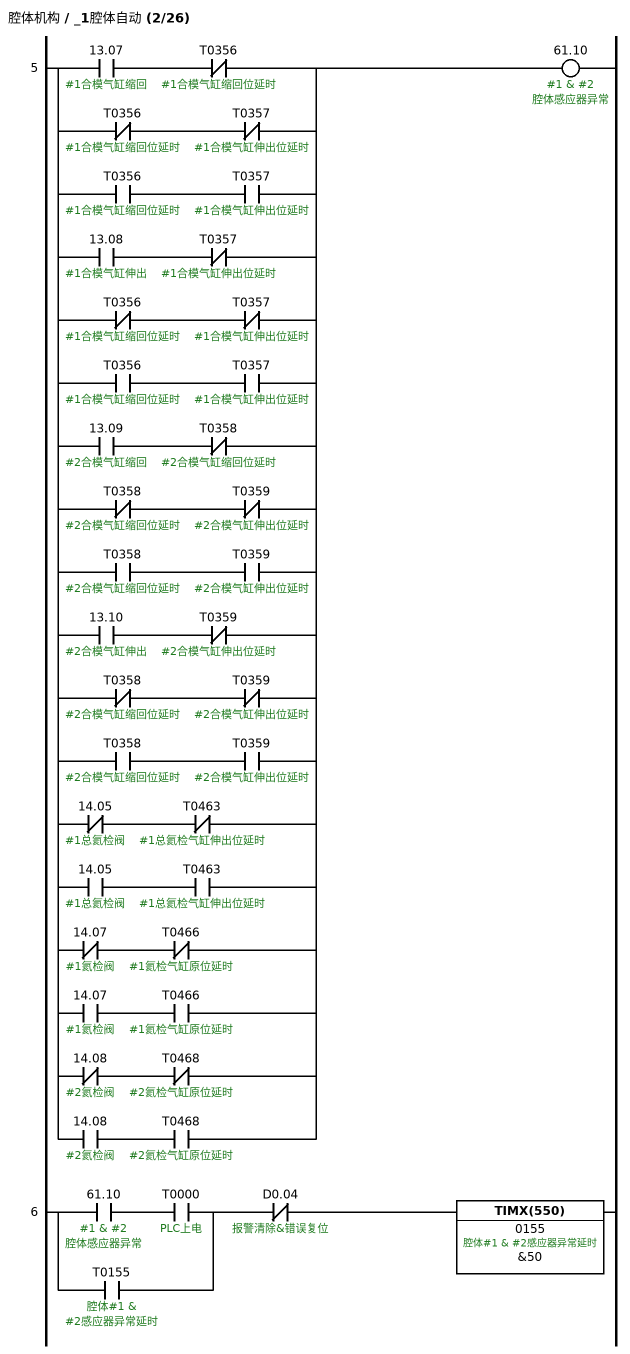
; [picture p240: 腔体机构 / _1腔体自动, rungs 5-6]
; rung 5
LD 13.07  ; #1合模气缸缩回
ANDNOT T0356  ; #1合模气缸缩回位延时
LDNOT T0356  ; #1合模气缸缩回位延时
ANDNOT T0357  ; #1合模气缸伸出位延时
ORLD
LD T0356  ; #1合模气缸缩回位延时
AND T0357  ; #1合模气缸伸出位延时
ORLD
LD 13.08  ; #1合模气缸伸出
ANDNOT T0357  ; #1合模气缸伸出位延时
ORLD
LDNOT T0356  ; #1合模气缸缩回位延时
ANDNOT T0357  ; #1合模气缸伸出位延时
ORLD
LD T0356  ; #1合模气缸缩回位延时
AND T0357  ; #1合模气缸伸出位延时
ORLD
LD 13.09  ; #2合模气缸缩回
ANDNOT T0358  ; #2合模气缸缩回位延时
ORLD
LDNOT T0358  ; #2合模气缸缩回位延时
ANDNOT T0359  ; #2合模气缸伸出位延时
ORLD
LD T0358  ; #2合模气缸缩回位延时
AND T0359  ; #2合模气缸伸出位延时
ORLD
LD 13.10  ; #2合模气缸伸出
ANDNOT T0359  ; #2合模气缸伸出位延时
ORLD
LDNOT T0358  ; #2合模气缸缩回位延时
ANDNOT T0359  ; #2合模气缸伸出位延时
ORLD
LD T0358  ; #2合模气缸缩回位延时
AND T0359  ; #2合模气缸伸出位延时
ORLD
LDNOT 14.05  ; #1总氦检阀
ANDNOT T0463  ; #1总氦检气缸伸出位延时
ORLD
LD 14.05  ; #1总氦检阀
AND T0463  ; #1总氦检气缸伸出位延时
ORLD
LDNOT 14.07  ; #1氦检阀
ANDNOT T0466  ; #1氦检气缸原位延时
ORLD
LD 14.07  ; #1氦检阀
AND T0466  ; #1氦检气缸原位延时
ORLD
LDNOT 14.08  ; #2氦检阀
ANDNOT T0468  ; #2氦检气缸原位延时
ORLD
LD 14.08  ; #2氦检阀
AND T0468  ; #2氦检气缸原位延时
ORLD
OUT 61.10  ; #1 & #2 腔体感应器异常
; rung 6
LD 61.10  ; #1 & #2 腔体感应器异常
AND T0000  ; PLC上电
OR T0155  ; 腔体#1 & #2感应器异常延时
ANDNOT D0.04  ; 报警清除&错误复位
TIMX(550) 0155 &50  ; 腔体#1 & #2感应器异常延时

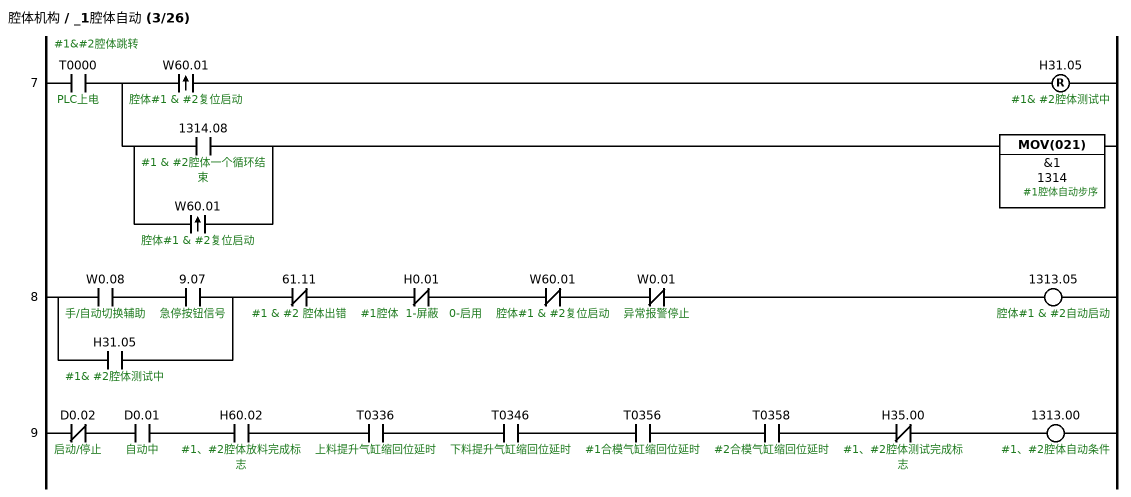
; rung 7: #1&#2腔体跳转
LD T0000  ; PLC上电
OUT TR0
@AND W60.01  ; 腔体#1 & #2复位启动
RSET H31.05  ; #1& #2腔体测试中
LD TR0
LD 1314.08  ; #1 & #2腔体一个循环结束
@OR W60.01  ; 腔体#1 & #2复位启动
ANDLD
MOV(021) &1 1314  ; #1腔体自动步序
; rung 8
LD W0.08  ; 手/自动切换辅助
AND 9.07  ; 急停按钮信号
OR H31.05  ; #1& #2腔体测试中
ANDNOT 61.11  ; #1 & #2 腔体出错
ANDNOT H0.01  ; #1腔体  1-屏蔽   0-启用
ANDNOT W60.01  ; 腔体#1 & #2复位启动
ANDNOT W0.01  ; 异常报警停止
OUT 1313.05  ; 腔体#1 & #2自动启动
; rung 9
LDNOT D0.02  ; 启动/停止
AND D0.01  ; 自动中
AND H60.02  ; #1、#2腔体放料完成标志
AND T0336  ; 上料提升气缸缩回位延时
AND T0346  ; 下料提升气缸缩回位延时
AND T0356  ; #1合模气缸缩回位延时
AND T0358  ; #2合模气缸缩回位延时
ANDNOT H35.00  ; #1、#2腔体测试完成标志
OUT 1313.00  ; #1、#2腔体自动条件

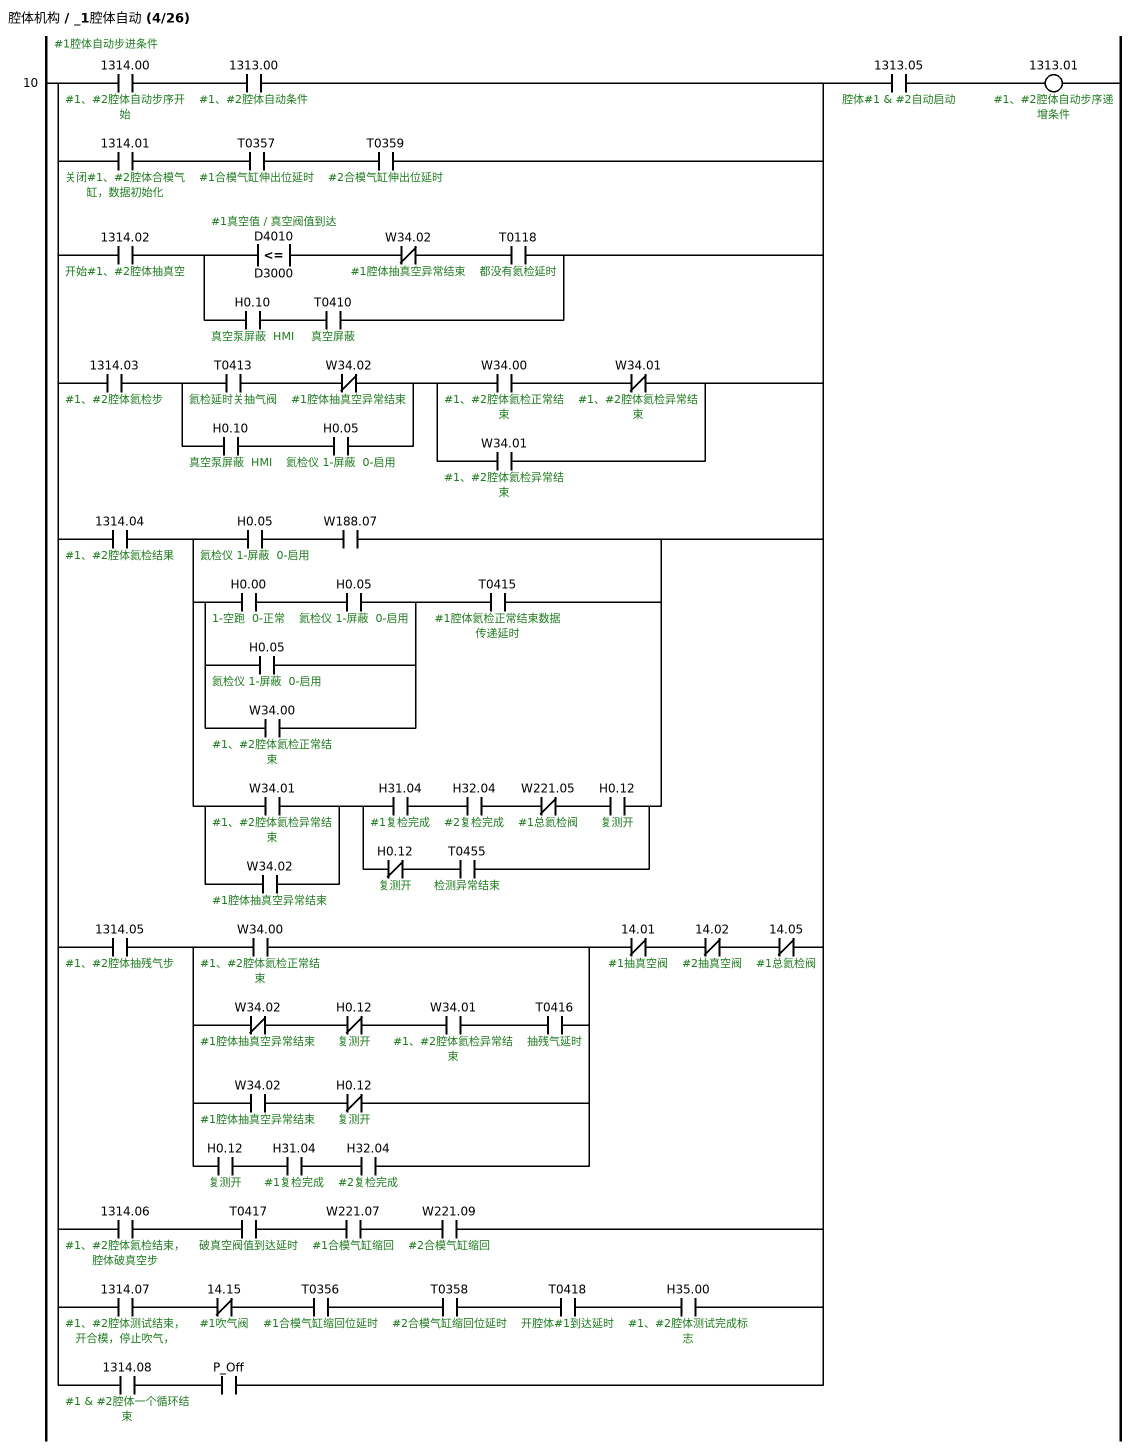
; rung 10: #1腔体自动步进条件
LD 1314.00  ; #1、#2腔体自动步序开始
AND 1313.00  ; #1、#2腔体自动条件
LD 1314.01  ; 关闭#1、#2腔体合模气缸，数据初始化
AND T0357  ; #1合模气缸伸出位延时
AND T0359  ; #2合模气缸伸出位延时
ORLD
LD 1314.02  ; 开始#1、#2腔体抽真空
LD<=F(332) D4010 D3000  ; #1真空值, 真空阀值到达
ANDNOT W34.02  ; #1腔体抽真空异常结束
AND T0118  ; 都没有氦检延时
LD H0.10  ; 真空泵屏蔽  HMI
AND T0410  ; 真空屏蔽
ORLD
ANDLD
ORLD
LD 1314.03  ; #1、#2腔体氦检步
LD T0413  ; 氦检延时关抽气阀
ANDNOT W34.02  ; #1腔体抽真空异常结束
LD H0.10  ; 真空泵屏蔽  HMI
AND H0.05  ; 氦检仪 1-屏蔽  0-启用
ORLD
ANDLD
LD W34.00  ; #1、#2腔体氦检正常结束
ANDNOT W34.01  ; #1、#2腔体氦检异常结束
OR W34.01  ; #1、#2腔体氦检异常结束
ANDLD
ORLD
LD 1314.04  ; #1、#2腔体氦检结果
LD H0.05  ; 氦检仪 1-屏蔽  0-启用
AND W188.07
LD H0.00  ; 1-空跑  0-正常
AND H0.05  ; 氦检仪 1-屏蔽  0-启用
OR H0.05  ; 氦检仪 1-屏蔽  0-启用
OR W34.00  ; #1、#2腔体氦检正常结束
AND T0415  ; #1腔体氦检正常结束数据传递延时
ORLD
LD W34.01  ; #1、#2腔体氦检异常结束
OR W34.02  ; #1腔体抽真空异常结束
LD H31.04  ; #1复检完成
AND H32.04  ; #2复检完成
ANDNOT W221.05  ; #1总氦检阀
AND H0.12  ; 复测开
LDNOT H0.12  ; 复测开
AND T0455  ; 检测异常结束
ORLD
ANDLD
ORLD
ANDLD
ORLD
LD 1314.05  ; #1、#2腔体抽残气步
LD W34.00  ; #1、#2腔体氦检正常结束
LDNOT W34.02  ; #1腔体抽真空异常结束
ANDNOT H0.12  ; 复测开
AND W34.01  ; #1、#2腔体氦检异常结束
AND T0416  ; 抽残气延时
ORLD
LD W34.02  ; #1腔体抽真空异常结束
ANDNOT H0.12  ; 复测开
ORLD
LD H0.12  ; 复测开
AND H31.04  ; #1复检完成
AND H32.04  ; #2复检完成
ORLD
ANDLD
ANDNOT 14.01  ; #1抽真空阀
ANDNOT 14.02  ; #2抽真空阀
ANDNOT 14.05  ; #1总氦检阀
ORLD
LD 1314.06  ; #1、#2腔体氦检结束，腔体破真空步
AND T0417  ; 破真空阀值到达延时
AND W221.07  ; #1合模气缸缩回
AND W221.09  ; #2合模气缸缩回
ORLD
LD 1314.07  ; #1、#2腔体测试结束，开合模，停止吹气，
ANDNOT 14.15  ; #1吹气阀
AND T0356  ; #1合模气缸缩回位延时
AND T0358  ; #2合模气缸缩回位延时
AND T0418  ; 开腔体#1到达延时
AND H35.00  ; #1、#2腔体测试完成标志
ORLD
LD 1314.08  ; #1 & #2腔体一个循环结束
AND P_Off
ORLD
AND 1313.05  ; 腔体#1 & #2自动启动
OUT 1313.01  ; #1、#2腔体自动步序递增条件

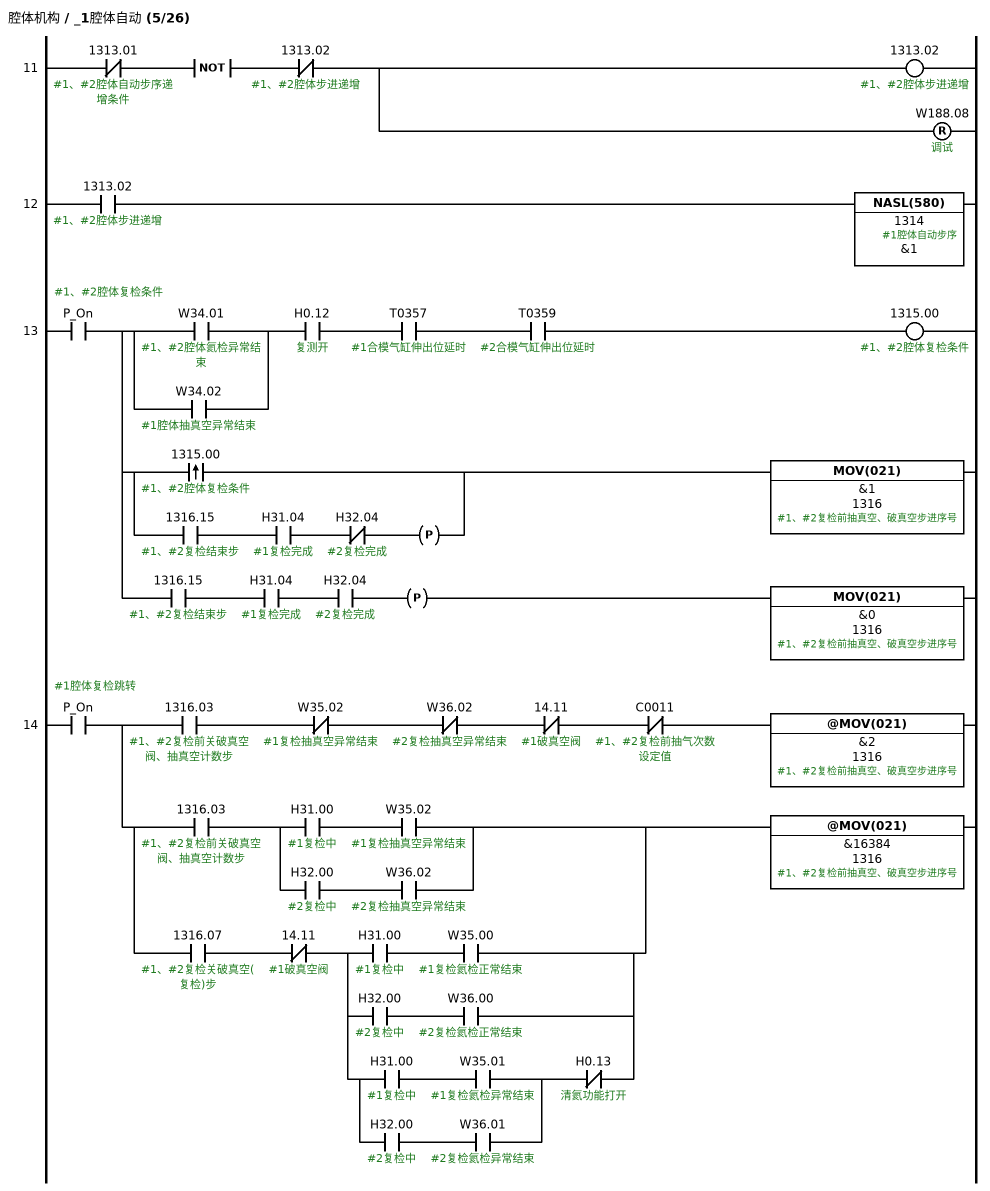
; rung 11
LDNOT 1313.01  ; #1、#2腔体自动步序递增条件
NOT(520)
ANDNOT 1313.02  ; #1、#2腔体步进递增
OUT 1313.02  ; #1、#2腔体步进递增
RSET W188.08  ; 调试
; rung 12
LD 1313.02  ; #1、#2腔体步进递增
NASL(580) 1314 &1  ; #1腔体自动步序
; rung 13: #1、#2腔体复检条件
LD P_On
OUT TR0
LD W34.01  ; #1、#2腔体氦检异常结束
OR W34.02  ; #1腔体抽真空异常结束
ANDLD
AND H0.12  ; 复测开
AND T0357  ; #1合模气缸伸出位延时
AND T0359  ; #2合模气缸伸出位延时
OUT 1315.00  ; #1、#2腔体复检条件
LD TR0
@LD 1315.00  ; #1、#2腔体复检条件
LD 1316.15  ; #1、#2复检结束步
AND H31.04  ; #1复检完成
ANDNOT H32.04  ; #2复检完成
UP(521)
ORLD
ANDLD
MOV(021) &1 1316  ; #1、#2复检前抽真空、破真空步进序号
LD TR0
AND 1316.15  ; #1、#2复检结束步
AND H31.04  ; #1复检完成
AND H32.04  ; #2复检完成
UP(521)
MOV(021) &0 1316  ; #1、#2复检前抽真空、破真空步进序号
; rung 14: #1腔体复检跳转
LD P_On
OUT TR0
AND 1316.03  ; #1、#2复检前关破真空阀、抽真空计数步
ANDNOT W35.02  ; #1复检抽真空异常结束
ANDNOT W36.02  ; #2复检抽真空异常结束
ANDNOT 14.11  ; #1破真空阀
ANDNOT C0011  ; #1、#2复检前抽气次数设定值
@MOV(021) &2 1316  ; #1、#2复检前抽真空、破真空步进序号
LD TR0
LD 1316.03  ; #1、#2复检前关破真空阀、抽真空计数步
LD H31.00  ; #1复检中
AND W35.02  ; #1复检抽真空异常结束
LD H32.00  ; #2复检中
AND W36.02  ; #2复检抽真空异常结束
ORLD
ANDLD
LD 1316.07  ; #1、#2复检关破真空(复检)步
ANDNOT 14.11  ; #1破真空阀
LD H31.00  ; #1复检中
AND W35.00  ; #1复检氦检正常结束
LD H32.00  ; #2复检中
AND W36.00  ; #2复检氦检正常结束
ORLD
LD H31.00  ; #1复检中
AND W35.01  ; #1复检氦检异常结束
LD H32.00  ; #2复检中
AND W36.01  ; #2复检氦检异常结束
ORLD
ANDNOT H0.13  ; 清氦功能打开
ORLD
ANDLD
ORLD
ANDLD
@MOV(021) &16384 1316  ; #1、#2复检前抽真空、破真空步进序号

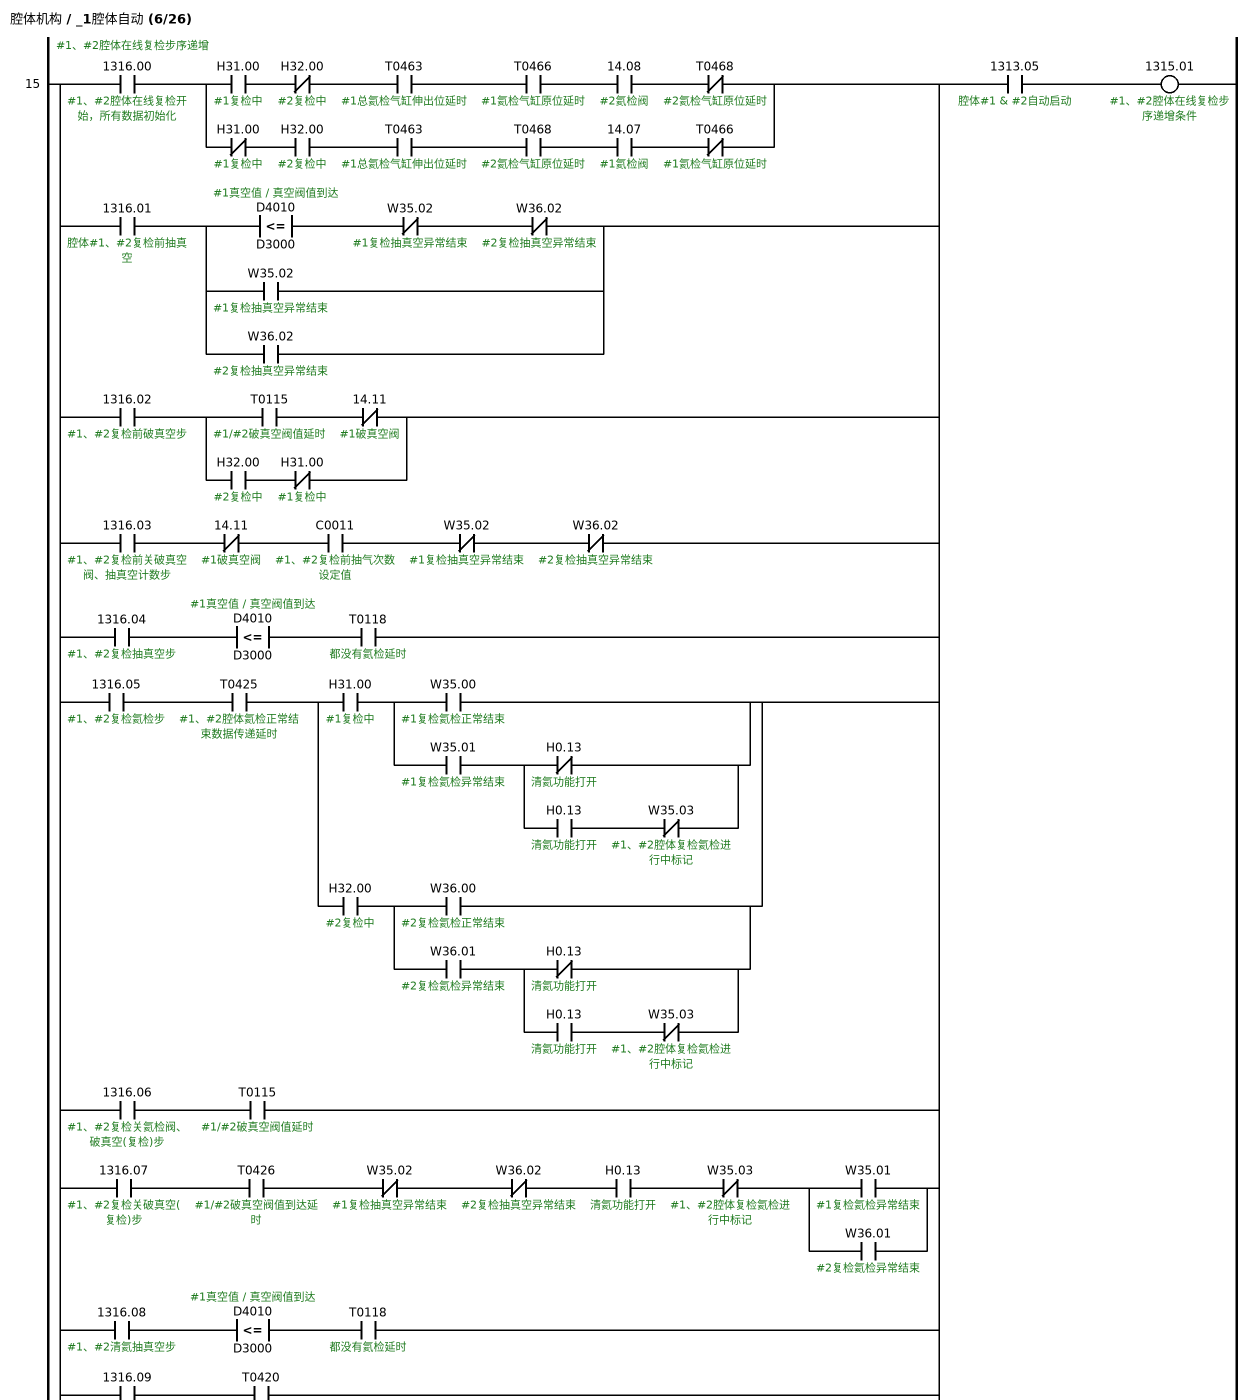

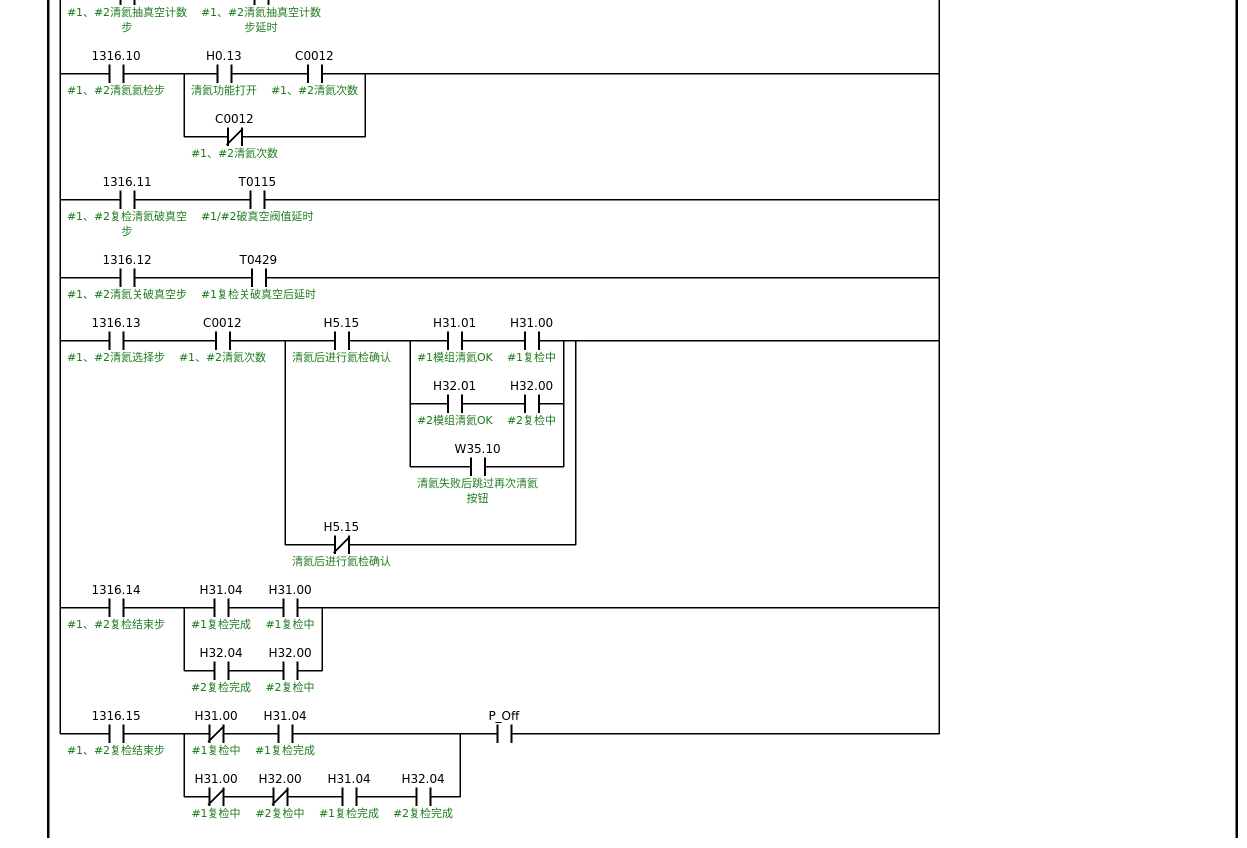
; rung 15: #1、#2腔体在线复检步序递增
LD 1316.00  ; #1、#2腔体在线复检开始，所有数据初始化
LD H31.00  ; #1复检中
ANDNOT H32.00  ; #2复检中
AND T0463  ; #1总氦检气缸伸出位延时
AND T0466  ; #1氦检气缸原位延时
AND 14.08  ; #2氦检阀
ANDNOT T0468  ; #2氦检气缸原位延时
LDNOT H31.00  ; #1复检中
AND H32.00  ; #2复检中
AND T0463  ; #1总氦检气缸伸出位延时
AND T0468  ; #2氦检气缸原位延时
AND 14.07  ; #1氦检阀
ANDNOT T0466  ; #1氦检气缸原位延时
ORLD
ANDLD
LD 1316.01  ; 腔体#1、#2复检前抽真空
LD<=F(332) D4010 D3000  ; #1真空值, 真空阀值到达
ANDNOT W35.02  ; #1复检抽真空异常结束
ANDNOT W36.02  ; #2复检抽真空异常结束
OR W35.02  ; #1复检抽真空异常结束
OR W36.02  ; #2复检抽真空异常结束
ANDLD
ORLD
LD 1316.02  ; #1、#2复检前破真空步
LD T0115  ; #1/#2破真空阀值延时
ANDNOT 14.11  ; #1破真空阀
LD H32.00  ; #2复检中
ANDNOT H31.00  ; #1复检中
ORLD
ANDLD
ORLD
LD 1316.03  ; #1、#2复检前关破真空阀、抽真空计数步
ANDNOT 14.11  ; #1破真空阀
AND C0011  ; #1、#2复检前抽气次数设定值
ANDNOT W35.02  ; #1复检抽真空异常结束
ANDNOT W36.02  ; #2复检抽真空异常结束
ORLD
LD 1316.04  ; #1、#2复检抽真空步
AND<=F(332) D4010 D3000  ; #1真空值, 真空阀值到达
AND T0118  ; 都没有氦检延时
ORLD
LD 1316.05  ; #1、#2复检氦检步
AND T0425  ; #1、#2腔体氦检正常结束数据传递延时
LD H31.00  ; #1复检中
LD W35.00  ; #1复检氦检正常结束
LD W35.01  ; #1复检氦检异常结束
LDNOT H0.13  ; 清氦功能打开
LD H0.13  ; 清氦功能打开
ANDNOT W35.03  ; #1、#2腔体复检氦检进行中标记
ORLD
ANDLD
ORLD
ANDLD
LD H32.00  ; #2复检中
LD W36.00  ; #2复检氦检正常结束
LD W36.01  ; #2复检氦检异常结束
LDNOT H0.13  ; 清氦功能打开
LD H0.13  ; 清氦功能打开
ANDNOT W35.03  ; #1、#2腔体复检氦检进行中标记
ORLD
ANDLD
ORLD
ANDLD
ORLD
ANDLD
ORLD
LD 1316.06  ; #1、#2复检关氦检阀、破真空(复检)步
AND T0115  ; #1/#2破真空阀值延时
ORLD
LD 1316.07  ; #1、#2复检关破真空(复检)步
AND T0426  ; #1/#2破真空阀值到达延时
ANDNOT W35.02  ; #1复检抽真空异常结束
ANDNOT W36.02  ; #2复检抽真空异常结束
AND H0.13  ; 清氦功能打开
ANDNOT W35.03  ; #1、#2腔体复检氦检进行中标记
LD W35.01  ; #1复检氦检异常结束
OR W36.01  ; #2复检氦检异常结束
ANDLD
ORLD
LD 1316.08  ; #1、#2清氦抽真空步
AND<=F(332) D4010 D3000  ; #1真空值, 真空阀值到达
AND T0118  ; 都没有氦检延时
ORLD
LD 1316.09  ; #1、#2清氦抽真空计数步
AND T0420  ; #1、#2清氦抽真空计数步延时
ORLD
LD 1316.10  ; #1、#2清氦氦检步
LD H0.13  ; 清氦功能打开
AND C0012  ; #1、#2清氦次数
ORNOT C0012  ; #1、#2清氦次数
ANDLD
ORLD
LD 1316.11  ; #1、#2复检清氦破真空步
AND T0115  ; #1/#2破真空阀值延时
ORLD
LD 1316.12  ; #1、#2清氦关破真空步
AND T0429  ; #1复检关破真空后延时
ORLD
LD 1316.13  ; #1、#2清氦选择步
AND C0012  ; #1、#2清氦次数
LD H5.15  ; 清氦后进行氦检确认
LD H31.01  ; #1模组清氦OK
AND H31.00  ; #1复检中
LD H32.01  ; #2模组清氦OK
AND H32.00  ; #2复检中
ORLD
OR W35.10  ; 清氦失败后跳过再次清氦按钮
ANDLD
ORNOT H5.15  ; 清氦后进行氦检确认
ANDLD
ORLD
LD 1316.14  ; #1、#2复检结束步
LD H31.04  ; #1复检完成
AND H31.00  ; #1复检中
LD H32.04  ; #2复检完成
AND H32.00  ; #2复检中
ORLD
ANDLD
ORLD
LD 1316.15  ; #1、#2复检结束步
LDNOT H31.00  ; #1复检中
AND H31.04  ; #1复检完成
LDNOT H31.00  ; #1复检中
ANDNOT H32.00  ; #2复检中
AND H31.04  ; #1复检完成
AND H32.04  ; #2复检完成
ORLD
ANDLD
AND P_Off
ORLD
AND 1313.05  ; 腔体#1 & #2自动启动
OUT 1315.01  ; #1、#2腔体在线复检步序递增条件

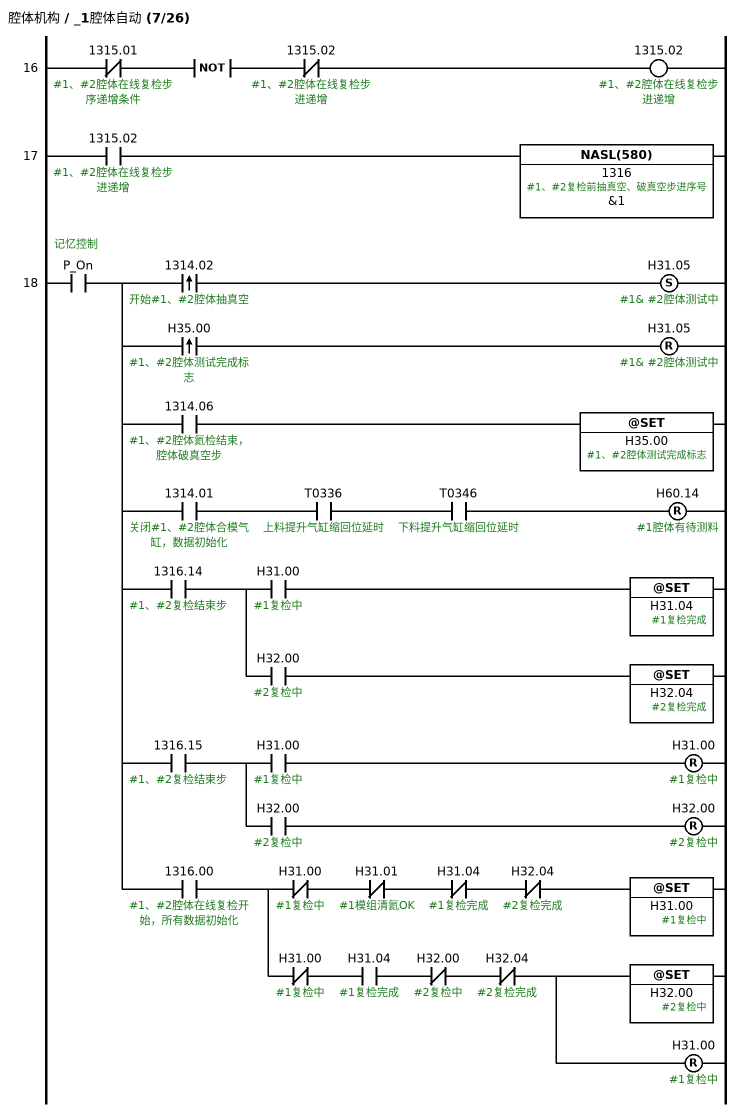
; rung 16
LDNOT 1315.01  ; #1、#2腔体在线复检步序递增条件
NOT(520)
ANDNOT 1315.02  ; #1、#2腔体在线复检步进递增
OUT 1315.02  ; #1、#2腔体在线复检步进递增
; rung 17
LD 1315.02  ; #1、#2腔体在线复检步进递增
NASL(580) 1316 &1  ; #1、#2复检前抽真空、破真空步进序号
; rung 18: 记忆控制
LD P_On
OUT TR0
@AND 1314.02  ; 开始#1、#2腔体抽真空
SET H31.05  ; #1& #2腔体测试中
LD TR0
@AND H35.00  ; #1、#2腔体测试完成标志
RSET H31.05  ; #1& #2腔体测试中
LD TR0
AND 1314.06  ; #1、#2腔体氦检结束，腔体破真空步
@SET H35.00  ; #1、#2腔体测试完成标志
LD TR0
AND 1314.01  ; 关闭#1、#2腔体合模气缸，数据初始化
AND T0336  ; 上料提升气缸缩回位延时
AND T0346  ; 下料提升气缸缩回位延时
RSET H60.14  ; #1腔体有待测料
LD TR0
AND 1316.14  ; #1、#2复检结束步
OUT TR1
AND H31.00  ; #1复检中
@SET H31.04  ; #1复检完成
LD TR1
AND H32.00  ; #2复检中
@SET H32.04  ; #2复检完成
LD TR0
AND 1316.15  ; #1、#2复检结束步
OUT TR1
AND H31.00  ; #1复检中
RSET H31.00  ; #1复检中
LD TR1
AND H32.00  ; #2复检中
RSET H32.00  ; #2复检中
LD TR0
AND 1316.00  ; #1、#2腔体在线复检开始，所有数据初始化
OUT TR0
ANDNOT H31.00  ; #1复检中
ANDNOT H31.01  ; #1模组清氦OK
ANDNOT H31.04  ; #1复检完成
ANDNOT H32.04  ; #2复检完成
@SET H31.00  ; #1复检中
LD TR0
ANDNOT H31.00  ; #1复检中
AND H31.04  ; #1复检完成
ANDNOT H32.00  ; #2复检中
ANDNOT H32.04  ; #2复检完成
@SET H32.00  ; #2复检中
RSET H31.00  ; #1复检中

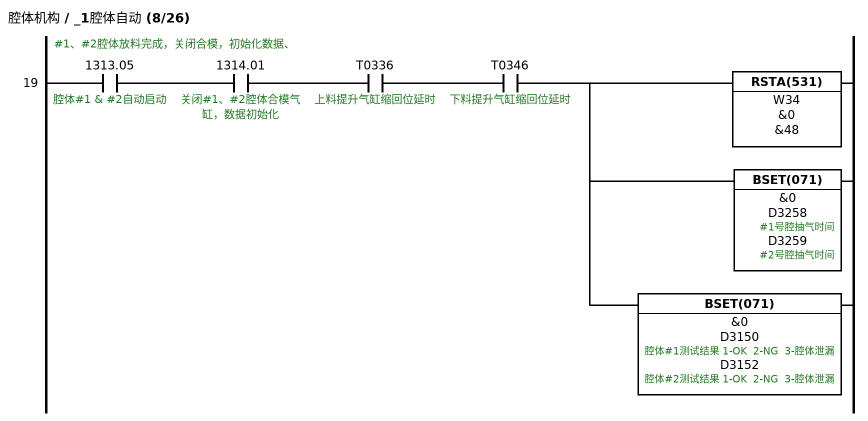
; rung 19: #1、#2腔体放料完成，关闭合模，初始化数据、
LD 1313.05  ; 腔体#1 & #2自动启动
AND 1314.01  ; 关闭#1、#2腔体合模气缸，数据初始化
AND T0336  ; 上料提升气缸缩回位延时
AND T0346  ; 下料提升气缸缩回位延时
RSTA(531) W34 &0 &48
BSET(071) &0 D3258 D3259  ; #1号腔抽气时间, #2号腔抽气时间
BSET(071) &0 D3150 D3152  ; 腔体#1测试结果 1-OK  2-NG  3-腔体泄漏, 腔体#2测试结果 1-OK  2-NG  3-腔体泄漏

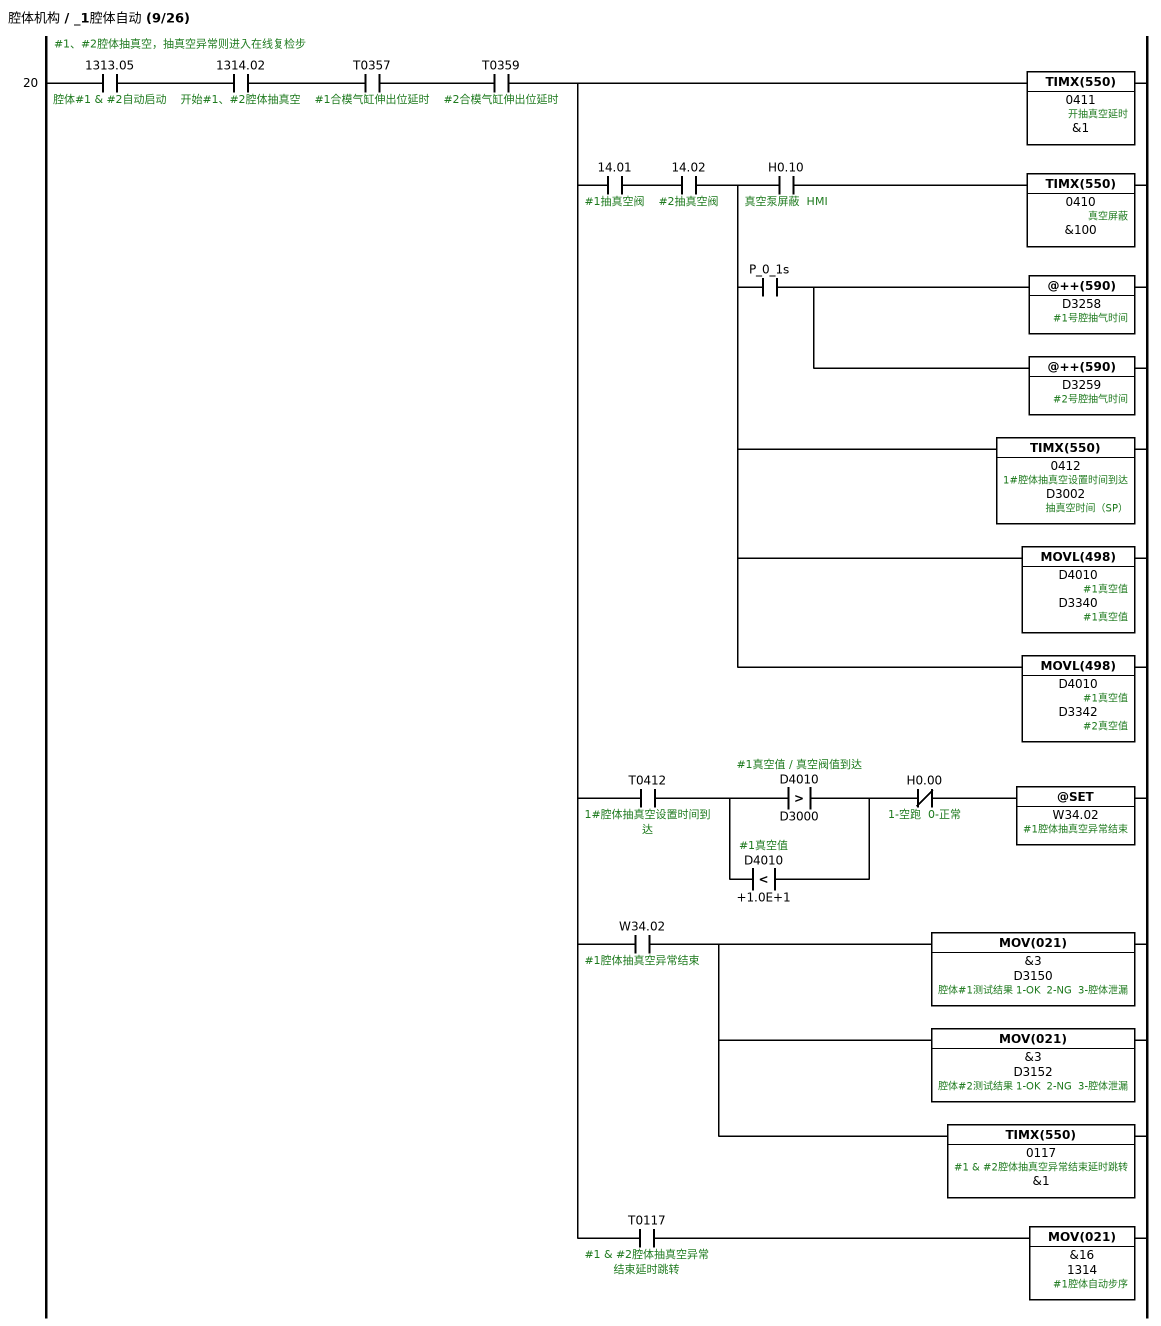
; rung 20: #1、#2腔体抽真空，抽真空异常则进入在线复检步
LD 1313.05  ; 腔体#1 & #2自动启动
AND 1314.02  ; 开始#1、#2腔体抽真空
AND T0357  ; #1合模气缸伸出位延时
AND T0359  ; #2合模气缸伸出位延时
OUT TR0
TIMX(550) 0411 &1  ; 开抽真空延时
AND 14.01  ; #1抽真空阀
AND 14.02  ; #2抽真空阀
OUT TR1
AND H0.10  ; 真空泵屏蔽  HMI
TIMX(550) 0410 &100  ; 真空屏蔽
LD TR1
AND P_0_1s
@++(590) D3258  ; #1号腔抽气时间
@++(590) D3259  ; #2号腔抽气时间
LD TR1
TIMX(550) 0412 D3002  ; 抽真空时间（SP）, 1#腔体抽真空设置时间到达
MOVL(498) D4010 D3340  ; #1真空值
MOVL(498) D4010 D3342  ; #1真空值, #2真空值
LD TR0
AND T0412  ; 1#腔体抽真空设置时间到达
LD>F(333) D4010 D3000  ; #1真空值, 真空阀值到达
OR<F(331) D4010 +1.0E+1  ; #1真空值
ANDLD
ANDNOT H0.00  ; 1-空跑  0-正常
@SET W34.02  ; #1腔体抽真空异常结束
LD TR0
AND W34.02  ; #1腔体抽真空异常结束
MOV(021) &3 D3150  ; 腔体#1测试结果 1-OK  2-NG  3-腔体泄漏
MOV(021) &3 D3152  ; 腔体#2测试结果 1-OK  2-NG  3-腔体泄漏
TIMX(550) 0117 &1  ; #1 & #2腔体抽真空异常结束延时跳转
LD TR0
AND T0117  ; #1 & #2腔体抽真空异常结束延时跳转
MOV(021) &16 1314  ; #1腔体自动步序

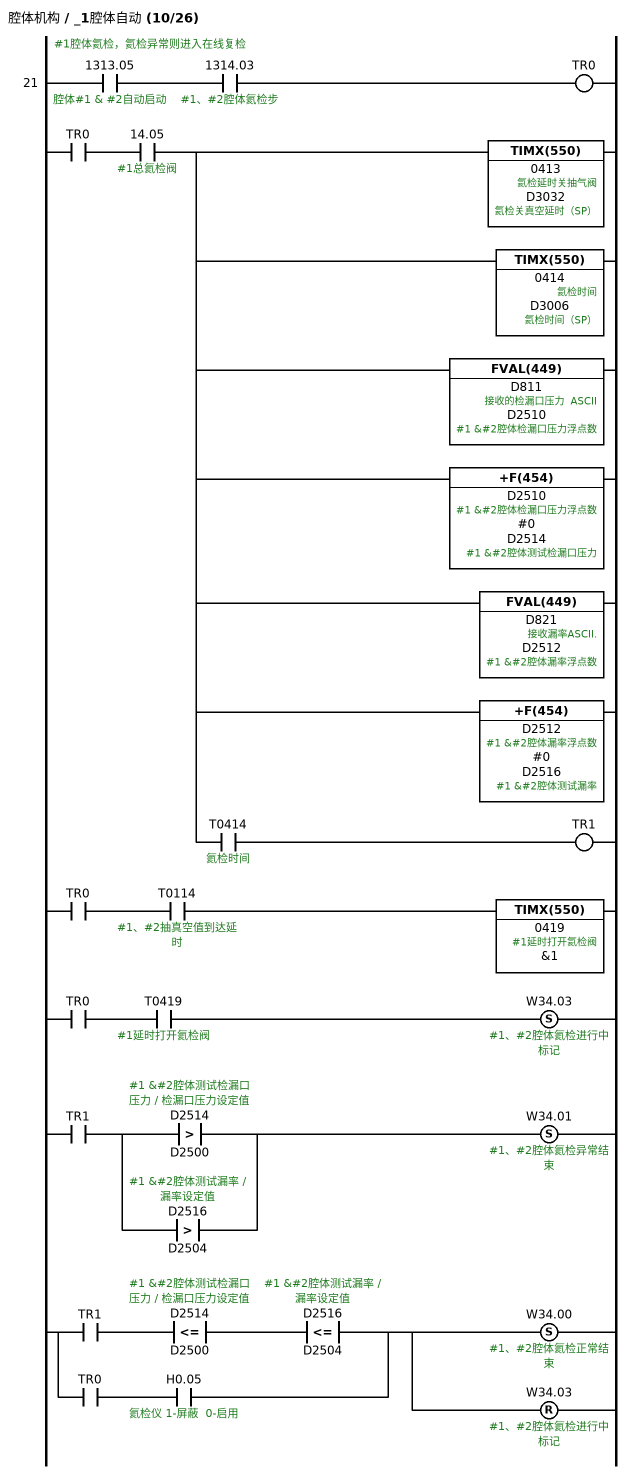
; rung 21: #1腔体氦检，氦检异常则进入在线复检
LD 1313.05  ; 腔体#1 & #2自动启动
AND 1314.03  ; #1、#2腔体氦检步
OUT TR0
AND T0114  ; #1、#2抽真空值到达延时
TIMX(550) 0419 &1  ; #1延时打开氦检阀
LD TR0
AND T0419  ; #1延时打开氦检阀
SET W34.03  ; #1、#2腔体氦检进行中标记
LD TR0
AND 14.05  ; #1总氦检阀
TIMX(550) 0413 D3032  ; 氦检关真空延时（SP）, 氦检延时关抽气阀
TIMX(550) 0414 D3006  ; 氦检时间（SP）, 氦检时间
FVAL(449) D811 D2510  ; 接收的检漏口压力  ASCII, #1 &#2腔体检漏口压力浮点数
+F(454) D2510 #0 D2514  ; #1 &#2腔体检漏口压力浮点数, #1 &#2腔体测试检漏口压力
FVAL(449) D821 D2512  ; 接收漏率ASCII., #1 &#2腔体漏率浮点数
+F(454) D2512 #0 D2516  ; #1 &#2腔体漏率浮点数, #1 &#2腔体测试漏率
AND T0414  ; 氦检时间
OUT TR1
LD>F(333) D2514 D2500  ; #1 &#2腔体测试检漏口压力, 检漏口压力设定值
OR>F(333) D2516 D2504  ; #1 &#2腔体测试漏率, 漏率设定值
ANDLD
SET W34.01  ; #1、#2腔体氦检异常结束
LD TR1
AND<=F(332) D2514 D2500  ; #1 &#2腔体测试检漏口压力, 检漏口压力设定值
AND<=F(332) D2516 D2504  ; #1 &#2腔体测试漏率, 漏率设定值
LD TR0
AND H0.05  ; 氦检仪 1-屏蔽  0-启用
ORLD
SET W34.00  ; #1、#2腔体氦检正常结束
RSET W34.03  ; #1、#2腔体氦检进行中标记

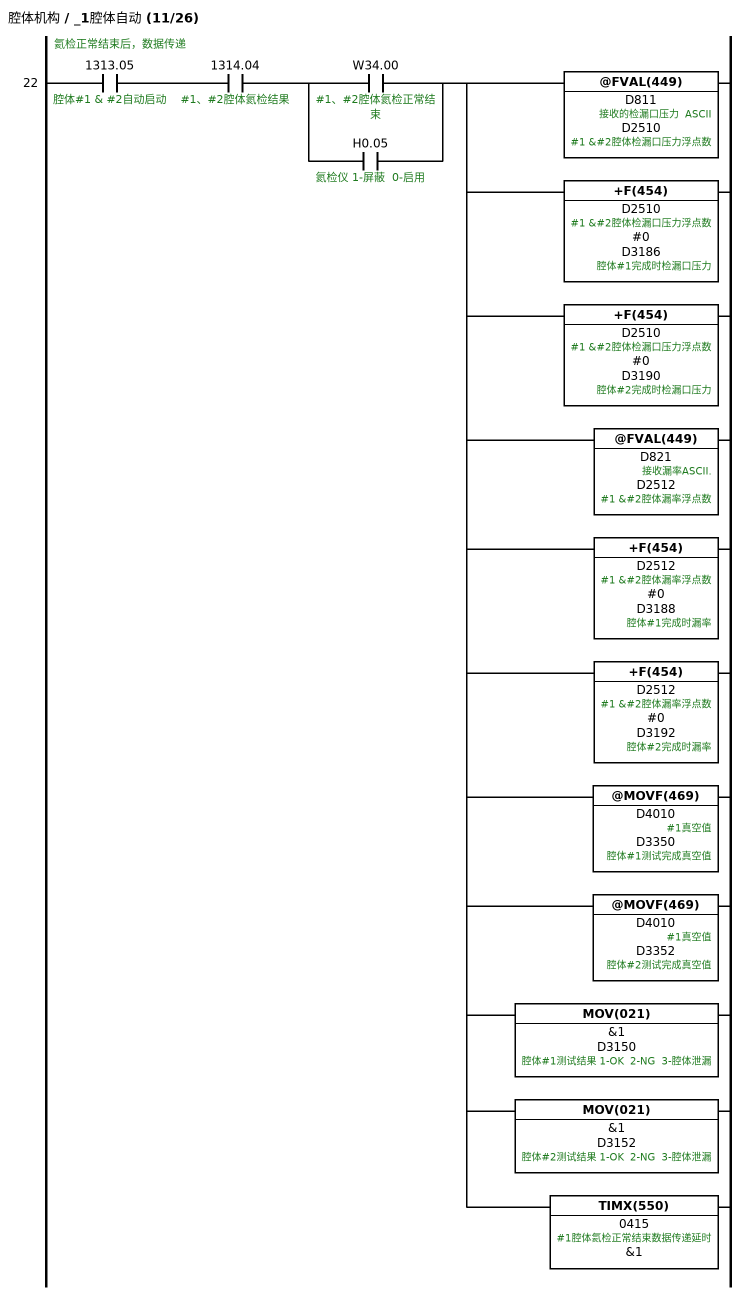
; rung 22: 氦检正常结束后，数据传递
LD 1313.05  ; 腔体#1 & #2自动启动
AND 1314.04  ; #1、#2腔体氦检结果
LD W34.00  ; #1、#2腔体氦检正常结束
OR H0.05  ; 氦检仪 1-屏蔽  0-启用
ANDLD
@FVAL(449) D811 D2510  ; 接收的检漏口压力  ASCII, #1 &#2腔体检漏口压力浮点数
+F(454) D2510 #0 D3186  ; #1 &#2腔体检漏口压力浮点数, 腔体#1完成时检漏口压力
+F(454) D2510 #0 D3190  ; #1 &#2腔体检漏口压力浮点数, 腔体#2完成时检漏口压力
@FVAL(449) D821 D2512  ; 接收漏率ASCII., #1 &#2腔体漏率浮点数
+F(454) D2512 #0 D3188  ; #1 &#2腔体漏率浮点数, 腔体#1完成时漏率
+F(454) D2512 #0 D3192  ; #1 &#2腔体漏率浮点数, 腔体#2完成时漏率
@MOVF(469) D4010 D3350  ; #1真空值, 腔体#1测试完成真空值
@MOVF(469) D4010 D3352  ; #1真空值, 腔体#2测试完成真空值
MOV(021) &1 D3150  ; 腔体#1测试结果 1-OK  2-NG  3-腔体泄漏
MOV(021) &1 D3152  ; 腔体#2测试结果 1-OK  2-NG  3-腔体泄漏
TIMX(550) 0415 &1  ; #1腔体氦检正常结束数据传递延时

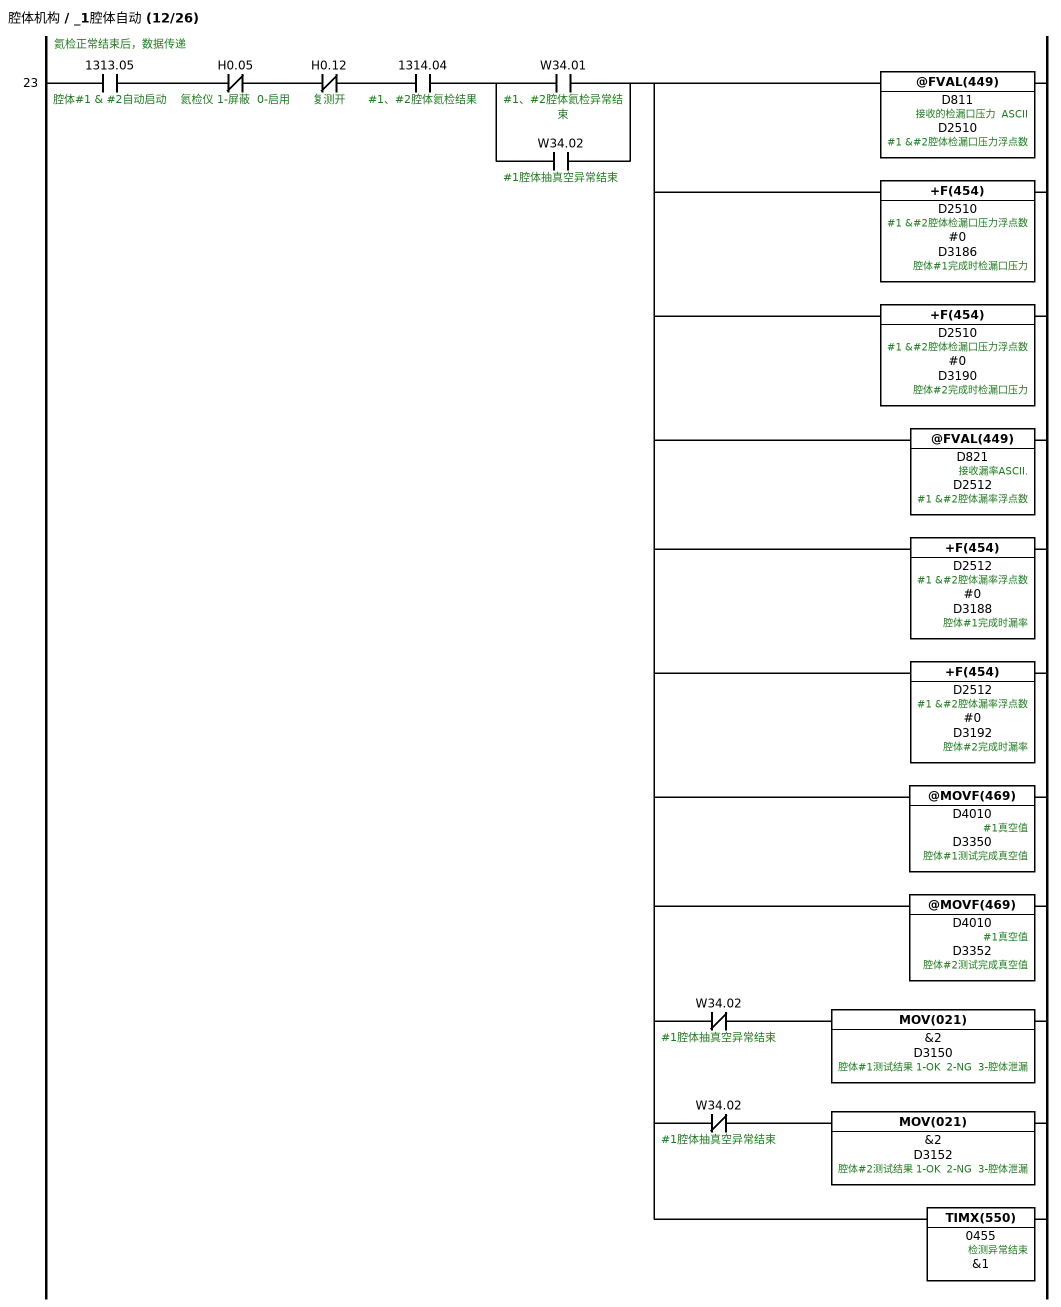
; rung 23: 氦检正常结束后，数据传递
LD 1313.05  ; 腔体#1 & #2自动启动
ANDNOT H0.05  ; 氦检仪 1-屏蔽  0-启用
ANDNOT H0.12  ; 复测开
AND 1314.04  ; #1、#2腔体氦检结果
LD W34.01  ; #1、#2腔体氦检异常结束
OR W34.02  ; #1腔体抽真空异常结束
ANDLD
OUT TR0
@FVAL(449) D811 D2510  ; 接收的检漏口压力  ASCII, #1 &#2腔体检漏口压力浮点数
+F(454) D2510 #0 D3186  ; #1 &#2腔体检漏口压力浮点数, 腔体#1完成时检漏口压力
+F(454) D2510 #0 D3190  ; #1 &#2腔体检漏口压力浮点数, 腔体#2完成时检漏口压力
@FVAL(449) D821 D2512  ; 接收漏率ASCII., #1 &#2腔体漏率浮点数
+F(454) D2512 #0 D3188  ; #1 &#2腔体漏率浮点数, 腔体#1完成时漏率
+F(454) D2512 #0 D3192  ; #1 &#2腔体漏率浮点数, 腔体#2完成时漏率
@MOVF(469) D4010 D3350  ; #1真空值, 腔体#1测试完成真空值
@MOVF(469) D4010 D3352  ; #1真空值, 腔体#2测试完成真空值
ANDNOT W34.02  ; #1腔体抽真空异常结束
MOV(021) &2 D3150  ; 腔体#1测试结果 1-OK  2-NG  3-腔体泄漏
LD TR0
ANDNOT W34.02  ; #1腔体抽真空异常结束
MOV(021) &2 D3152  ; 腔体#2测试结果 1-OK  2-NG  3-腔体泄漏
LD TR0
TIMX(550) 0455 &1  ; 检测异常结束

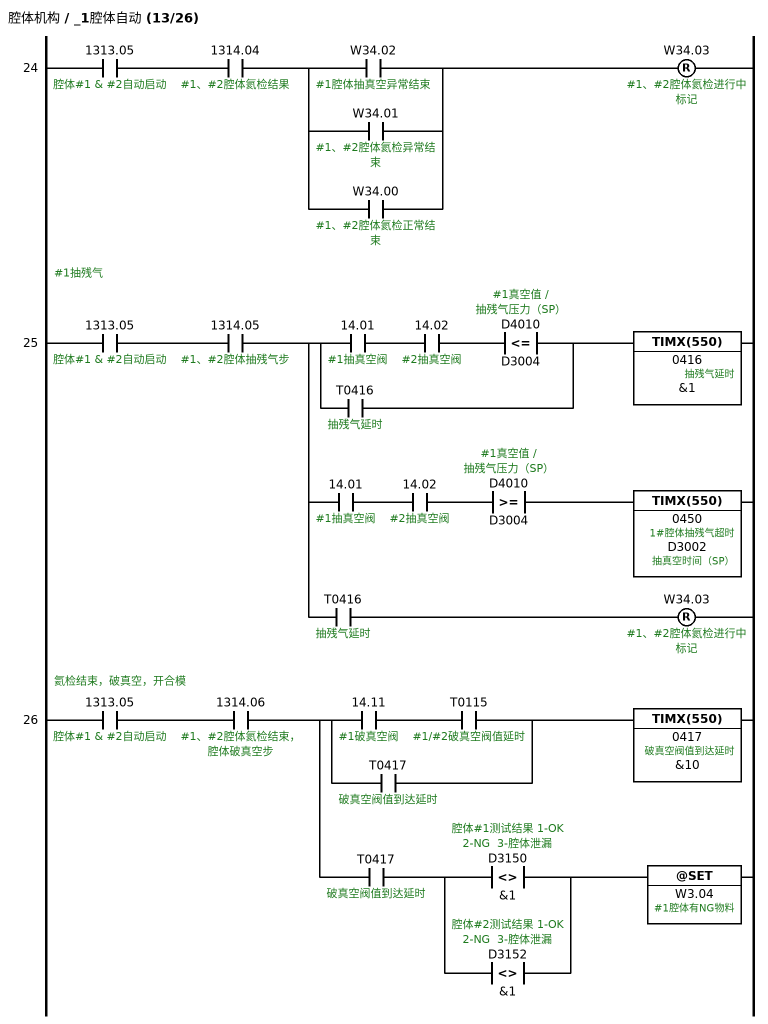
; rung 24
LD 1313.05  ; 腔体#1 & #2自动启动
AND 1314.04  ; #1、#2腔体氦检结果
LD W34.02  ; #1腔体抽真空异常结束
OR W34.01  ; #1、#2腔体氦检异常结束
OR W34.00  ; #1、#2腔体氦检正常结束
ANDLD
RSET W34.03  ; #1、#2腔体氦检进行中标记
; rung 25: #1抽残气
LD 1313.05  ; 腔体#1 & #2自动启动
AND 1314.05  ; #1、#2腔体抽残气步
OUT TR0
LD 14.01  ; #1抽真空阀
AND 14.02  ; #2抽真空阀
AND<=F(332) D4010 D3004  ; #1真空值, 抽残气压力（SP）
OR T0416  ; 抽残气延时
ANDLD
TIMX(550) 0416 &1  ; 抽残气延时
LD TR0
AND 14.01  ; #1抽真空阀
AND 14.02  ; #2抽真空阀
AND>=F(334) D4010 D3004  ; #1真空值, 抽残气压力（SP）
TIMX(550) 0450 D3002  ; 抽真空时间（SP）, 1#腔体抽残气超时
LD TR0
AND T0416  ; 抽残气延时
RSET W34.03  ; #1、#2腔体氦检进行中标记
; rung 26: 氦检结束，破真空，开合模
LD 1313.05  ; 腔体#1 & #2自动启动
AND 1314.06  ; #1、#2腔体氦检结束，腔体破真空步
OUT TR0
LD 14.11  ; #1破真空阀
AND T0115  ; #1/#2破真空阀值延时
OR T0417  ; 破真空阀值到达延时
ANDLD
TIMX(550) 0417 &10  ; 破真空阀值到达延时
LD TR0
AND T0417  ; 破真空阀值到达延时
LD<>(305) D3150 &1  ; 腔体#1测试结果 1-OK  2-NG  3-腔体泄漏
OR<>(305) D3152 &1  ; 腔体#2测试结果 1-OK  2-NG  3-腔体泄漏
ANDLD
@SET W3.04  ; #1腔体有NG物料

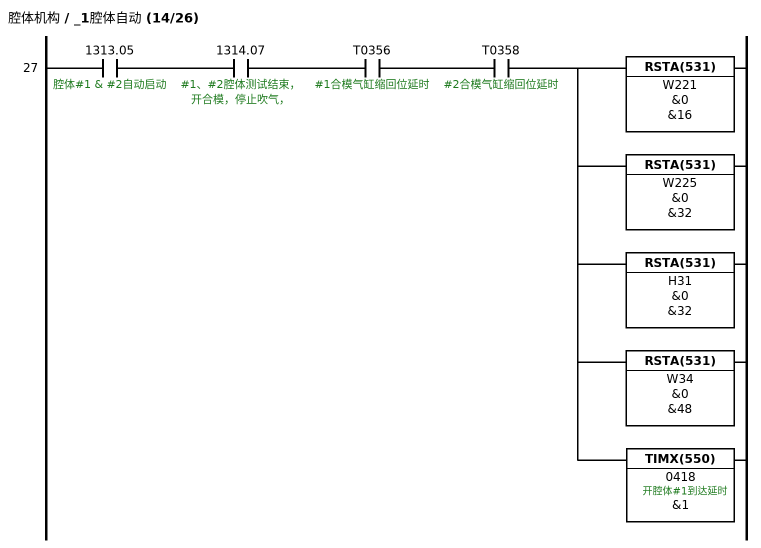
; rung 27
LD 1313.05  ; 腔体#1 & #2自动启动
AND 1314.07  ; #1、#2腔体测试结束，开合模，停止吹气，
AND T0356  ; #1合模气缸缩回位延时
AND T0358  ; #2合模气缸缩回位延时
RSTA(531) W221 &0 &16
RSTA(531) W225 &0 &32
RSTA(531) H31 &0 &32
RSTA(531) W34 &0 &48
TIMX(550) 0418 &1  ; 开腔体#1到达延时

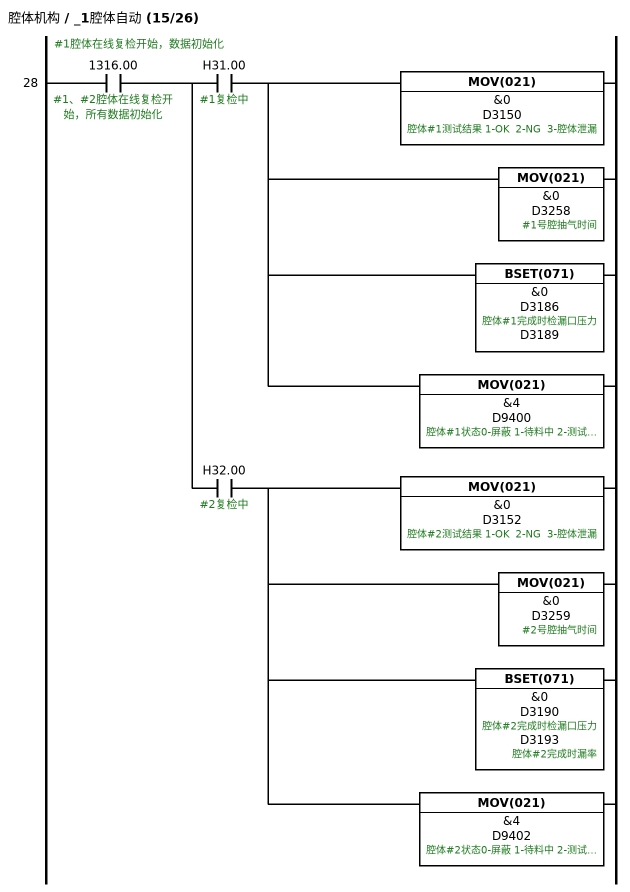
; rung 28: #1腔体在线复检开始，数据初始化
LD 1316.00  ; #1、#2腔体在线复检开始，所有数据初始化
OUT TR0
AND H31.00  ; #1复检中
MOV(021) &0 D3150  ; 腔体#1测试结果 1-OK  2-NG  3-腔体泄漏
MOV(021) &0 D3258  ; #1号腔抽气时间
BSET(071) &0 D3186 D3189  ; 腔体#1完成时检漏口压力
MOV(021) &4 D9400  ; 腔体#1状态0-屏蔽 1-待料中 2-测试中 3-测试完成 4-在线复检
LD TR0
AND H32.00  ; #2复检中
MOV(021) &0 D3152  ; 腔体#2测试结果 1-OK  2-NG  3-腔体泄漏
MOV(021) &0 D3259  ; #2号腔抽气时间
BSET(071) &0 D3190 D3193  ; 腔体#2完成时检漏口压力, 腔体#2完成时漏率
MOV(021) &4 D9402  ; 腔体#2状态0-屏蔽 1-待料中 2-测试中 3-测试完成 4-在线复检

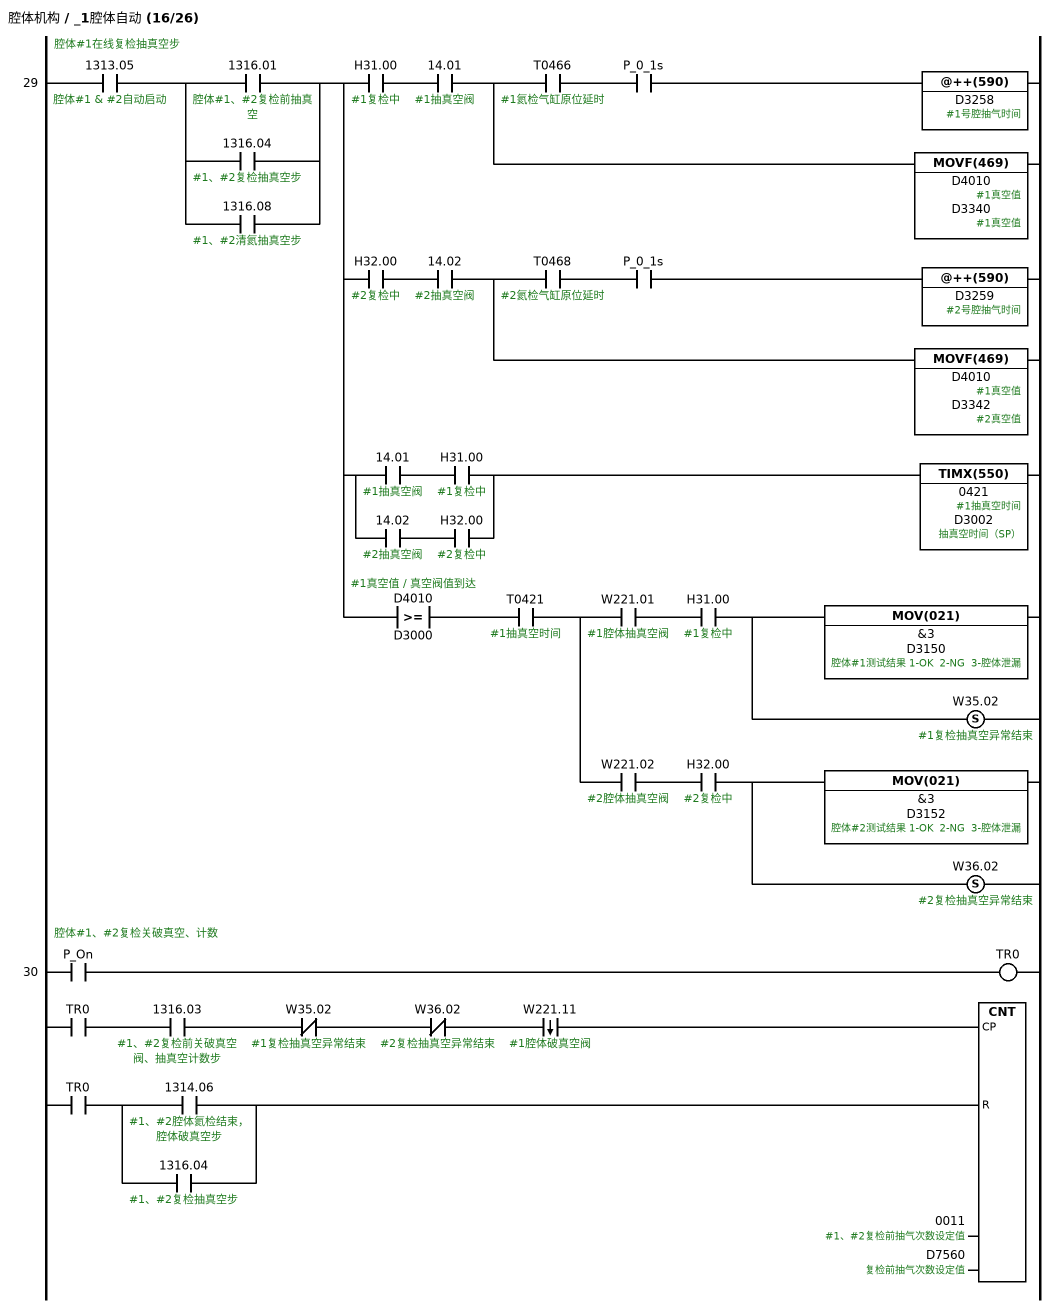
; rung 29: 腔体#1在线复检抽真空步
LD 1313.05  ; 腔体#1 & #2自动启动
LD 1316.01  ; 腔体#1、#2复检前抽真空
OR 1316.04  ; #1、#2复检抽真空步
OR 1316.08  ; #1、#2清氦抽真空步
ANDLD
OUT TR0
AND H31.00  ; #1复检中
AND 14.01  ; #1抽真空阀
OUT TR1
AND T0466  ; #1氦检气缸原位延时
AND P_0_1s
@++(590) D3258  ; #1号腔抽气时间
LD TR1
MOVF(469) D4010 D3340  ; #1真空值
LD TR0
AND H32.00  ; #2复检中
AND 14.02  ; #2抽真空阀
OUT TR1
AND T0468  ; #2氦检气缸原位延时
AND P_0_1s
@++(590) D3259  ; #2号腔抽气时间
LD TR1
MOVF(469) D4010 D3342  ; #1真空值, #2真空值
LD TR0
LD 14.01  ; #1抽真空阀
AND H31.00  ; #1复检中
LD 14.02  ; #2抽真空阀
AND H32.00  ; #2复检中
ORLD
ANDLD
TIMX(550) 0421 D3002  ; 抽真空时间（SP）, #1抽真空时间
LD TR0
AND>=F(334) D4010 D3000  ; #1真空值, 真空阀值到达
AND T0421  ; #1抽真空时间
OUT TR0
AND W221.01  ; #1腔体抽真空阀
AND H31.00  ; #1复检中
MOV(021) &3 D3150  ; 腔体#1测试结果 1-OK  2-NG  3-腔体泄漏
SET W35.02  ; #1复检抽真空异常结束
LD TR0
AND W221.02  ; #2腔体抽真空阀
AND H32.00  ; #2复检中
MOV(021) &3 D3152  ; 腔体#2测试结果 1-OK  2-NG  3-腔体泄漏
SET W36.02  ; #2复检抽真空异常结束
; rung 30: 腔体#1、#2复检关破真空、计数
LD P_On
OUT TR0
AND 1316.03  ; #1、#2复检前关破真空阀、抽真空计数步
ANDNOT W35.02  ; #1复检抽真空异常结束
ANDNOT W36.02  ; #2复检抽真空异常结束
%AND W221.11  ; #1腔体破真空阀
LD TR0
LD 1314.06  ; #1、#2腔体氦检结束，腔体破真空步
OR 1316.04  ; #1、#2复检抽真空步
ANDLD
CNT 0011 D7560  ; 复检前抽气次数设定值, #1、#2复检前抽气次数设定值

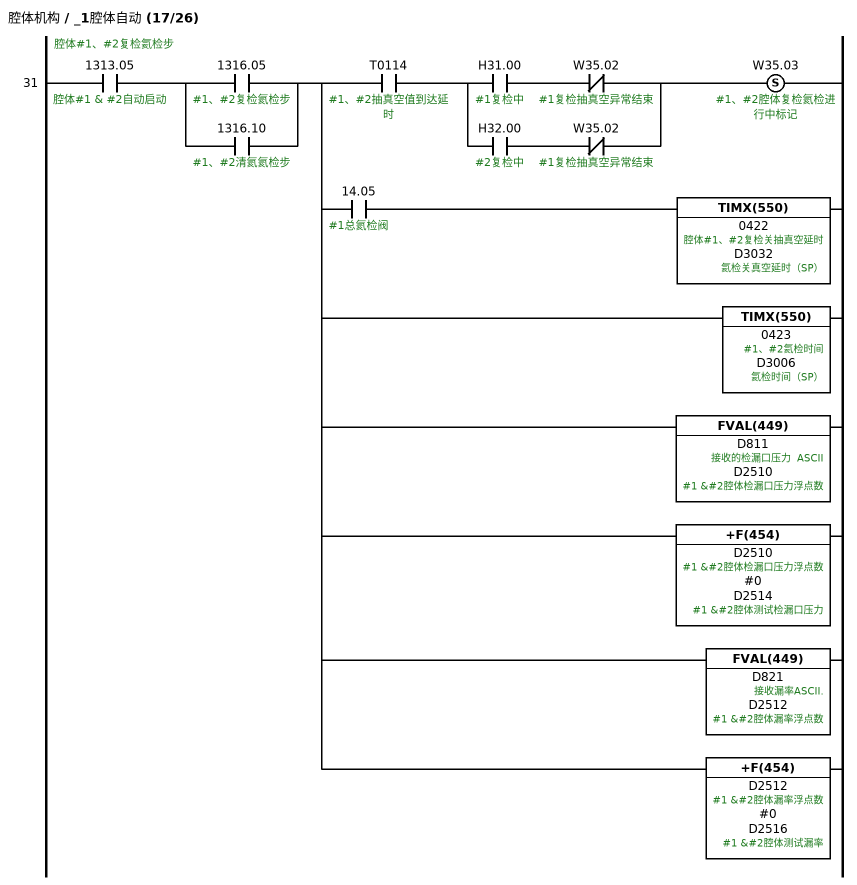
; rung 31: 腔体#1、#2复检氦检步
LD 1313.05  ; 腔体#1 & #2自动启动
LD 1316.05  ; #1、#2复检氦检步
OR 1316.10  ; #1、#2清氦氦检步
ANDLD
OUT TR0
AND T0114  ; #1、#2抽真空值到达延时
LD H31.00  ; #1复检中
ANDNOT W35.02  ; #1复检抽真空异常结束
LD H32.00  ; #2复检中
ANDNOT W35.02  ; #1复检抽真空异常结束
ORLD
ANDLD
SET W35.03  ; #1、#2腔体复检氦检进行中标记
LD TR0
AND 14.05  ; #1总氦检阀
TIMX(550) 0422 D3032  ; 氦检关真空延时（SP）, 腔体#1、#2复检关抽真空延时
LD TR0
TIMX(550) 0423 D3006  ; 氦检时间（SP）, #1、#2氦检时间
FVAL(449) D811 D2510  ; 接收的检漏口压力  ASCII, #1 &#2腔体检漏口压力浮点数
+F(454) D2510 #0 D2514  ; #1 &#2腔体检漏口压力浮点数, #1 &#2腔体测试检漏口压力
FVAL(449) D821 D2512  ; 接收漏率ASCII., #1 &#2腔体漏率浮点数
+F(454) D2512 #0 D2516  ; #1 &#2腔体漏率浮点数, #1 &#2腔体测试漏率

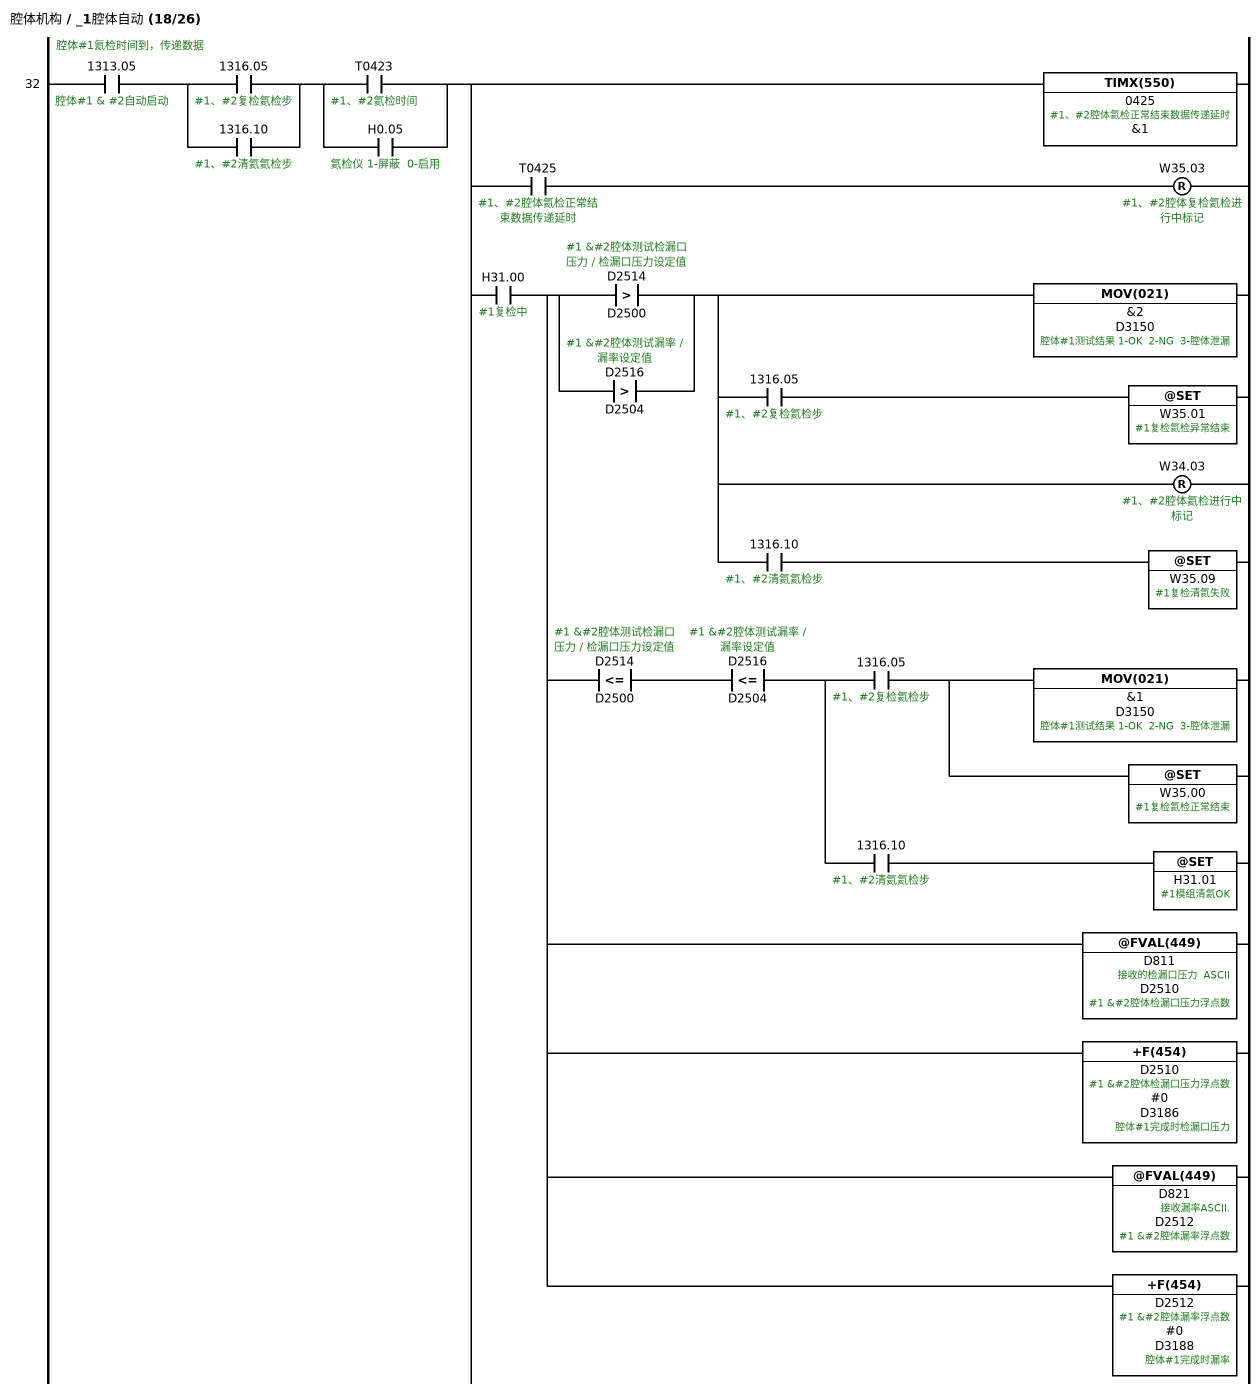

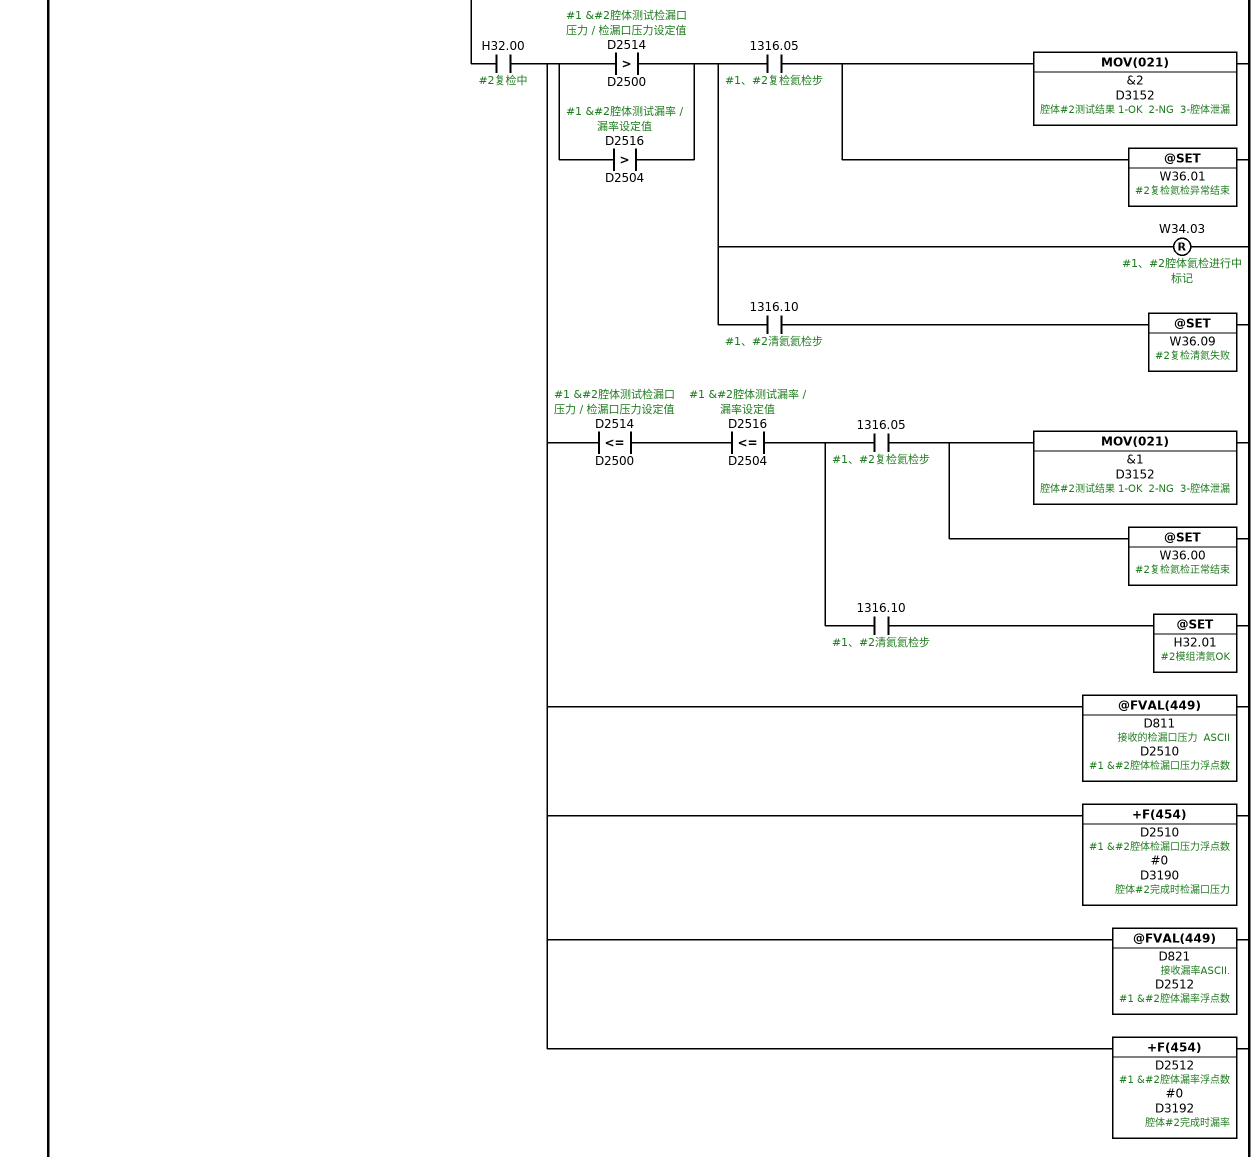
; rung 32: 腔体#1氦检时间到，传递数据
LD 1313.05  ; 腔体#1 & #2自动启动
LD 1316.05  ; #1、#2复检氦检步
OR 1316.10  ; #1、#2清氦氦检步
ANDLD
LD T0423  ; #1、#2氦检时间
OR H0.05  ; 氦检仪 1-屏蔽  0-启用
ANDLD
OUT TR0
TIMX(550) 0425 &1  ; #1、#2腔体氦检正常结束数据传递延时
AND T0425  ; #1、#2腔体氦检正常结束数据传递延时
RSET W35.03  ; #1、#2腔体复检氦检进行中标记
LD TR0
AND H31.00  ; #1复检中
OUT TR1
LD>F(333) D2514 D2500  ; #1 &#2腔体测试检漏口压力, 检漏口压力设定值
OR>F(333) D2516 D2504  ; #1 &#2腔体测试漏率, 漏率设定值
ANDLD
OUT TR2
MOV(021) &2 D3150  ; 腔体#1测试结果 1-OK  2-NG  3-腔体泄漏
AND 1316.05  ; #1、#2复检氦检步
@SET W35.01  ; #1复检氦检异常结束
LD TR2
RSET W34.03  ; #1、#2腔体氦检进行中标记
AND 1316.10  ; #1、#2清氦氦检步
@SET W35.09  ; #1复检清氦失败
LD TR1
AND<=F(332) D2514 D2500  ; #1 &#2腔体测试检漏口压力, 检漏口压力设定值
AND<=F(332) D2516 D2504  ; #1 &#2腔体测试漏率, 漏率设定值
OUT TR2
AND 1316.05  ; #1、#2复检氦检步
MOV(021) &1 D3150  ; 腔体#1测试结果 1-OK  2-NG  3-腔体泄漏
@SET W35.00  ; #1复检氦检正常结束
LD TR2
AND 1316.10  ; #1、#2清氦氦检步
@SET H31.01  ; #1模组清氦OK
LD TR1
@FVAL(449) D811 D2510  ; 接收的检漏口压力  ASCII, #1 &#2腔体检漏口压力浮点数
+F(454) D2510 #0 D3186  ; #1 &#2腔体检漏口压力浮点数, 腔体#1完成时检漏口压力
@FVAL(449) D821 D2512  ; 接收漏率ASCII., #1 &#2腔体漏率浮点数
+F(454) D2512 #0 D3188  ; #1 &#2腔体漏率浮点数, 腔体#1完成时漏率
LD TR0
AND H32.00  ; #2复检中
OUT TR0
LD>F(333) D2514 D2500  ; #1 &#2腔体测试检漏口压力, 检漏口压力设定值
OR>F(333) D2516 D2504  ; #1 &#2腔体测试漏率, 漏率设定值
ANDLD
OUT TR1
AND 1316.05  ; #1、#2复检氦检步
MOV(021) &2 D3152  ; 腔体#2测试结果 1-OK  2-NG  3-腔体泄漏
@SET W36.01  ; #2复检氦检异常结束
LD TR1
RSET W34.03  ; #1、#2腔体氦检进行中标记
AND 1316.10  ; #1、#2清氦氦检步
@SET W36.09  ; #2复检清氦失败
LD TR0
AND<=F(332) D2514 D2500  ; #1 &#2腔体测试检漏口压力, 检漏口压力设定值
AND<=F(332) D2516 D2504  ; #1 &#2腔体测试漏率, 漏率设定值
OUT TR1
AND 1316.05  ; #1、#2复检氦检步
MOV(021) &1 D3152  ; 腔体#2测试结果 1-OK  2-NG  3-腔体泄漏
@SET W36.00  ; #2复检氦检正常结束
LD TR1
AND 1316.10  ; #1、#2清氦氦检步
@SET H32.01  ; #2模组清氦OK
LD TR0
@FVAL(449) D811 D2510  ; 接收的检漏口压力  ASCII, #1 &#2腔体检漏口压力浮点数
+F(454) D2510 #0 D3190  ; #1 &#2腔体检漏口压力浮点数, 腔体#2完成时检漏口压力
@FVAL(449) D821 D2512  ; 接收漏率ASCII., #1 &#2腔体漏率浮点数
+F(454) D2512 #0 D3192  ; #1 &#2腔体漏率浮点数, 腔体#2完成时漏率

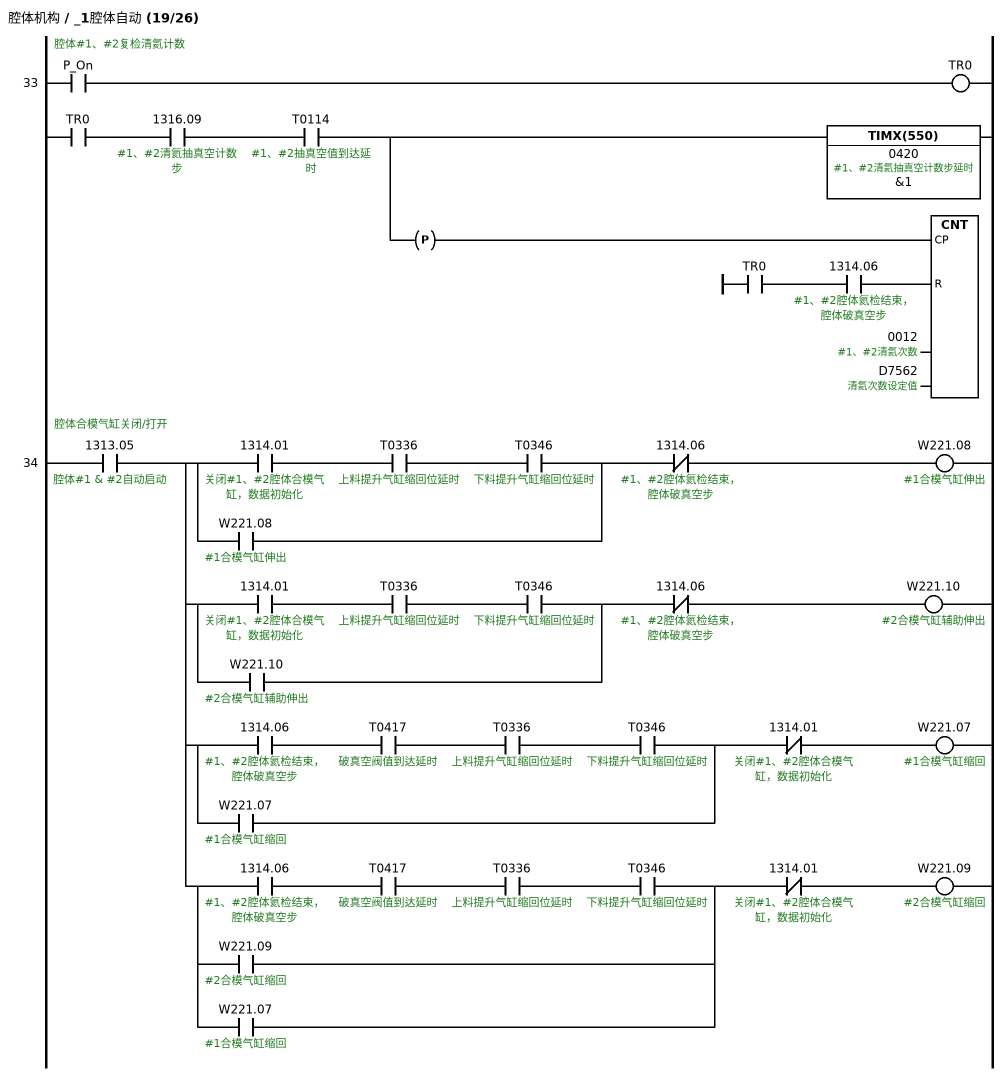
; rung 33: 腔体#1、#2复检清氦计数
LD P_On
OUT TR0
AND 1316.09  ; #1、#2清氦抽真空计数步
AND T0114  ; #1、#2抽真空值到达延时
TIMX(550) 0420 &1  ; #1、#2清氦抽真空计数步延时
UP(521)
LD TR0
AND 1314.06  ; #1、#2腔体氦检结束，腔体破真空步
CNT 0012 D7562  ; 清氦次数设定值, #1、#2清氦次数
; rung 34: 腔体合模气缸关闭/打开
LD 1313.05  ; 腔体#1 & #2自动启动
OUT TR0
LD 1314.01  ; 关闭#1、#2腔体合模气缸，数据初始化
AND T0336  ; 上料提升气缸缩回位延时
AND T0346  ; 下料提升气缸缩回位延时
OR W221.08  ; #1合模气缸伸出
ANDLD
ANDNOT 1314.06  ; #1、#2腔体氦检结束，腔体破真空步
OUT W221.08  ; #1合模气缸伸出
LD TR0
LD 1314.01  ; 关闭#1、#2腔体合模气缸，数据初始化
AND T0336  ; 上料提升气缸缩回位延时
AND T0346  ; 下料提升气缸缩回位延时
OR W221.10  ; #2合模气缸辅助伸出
ANDLD
ANDNOT 1314.06  ; #1、#2腔体氦检结束，腔体破真空步
OUT W221.10  ; #2合模气缸辅助伸出
LD TR0
LD 1314.06  ; #1、#2腔体氦检结束，腔体破真空步
AND T0417  ; 破真空阀值到达延时
AND T0336  ; 上料提升气缸缩回位延时
AND T0346  ; 下料提升气缸缩回位延时
OR W221.07  ; #1合模气缸缩回
ANDLD
ANDNOT 1314.01  ; 关闭#1、#2腔体合模气缸，数据初始化
OUT W221.07  ; #1合模气缸缩回
LD TR0
LD 1314.06  ; #1、#2腔体氦检结束，腔体破真空步
AND T0417  ; 破真空阀值到达延时
AND T0336  ; 上料提升气缸缩回位延时
AND T0346  ; 下料提升气缸缩回位延时
LD W221.09  ; #2合模气缸缩回
OR W221.07  ; #1合模气缸缩回
ORLD
ANDLD
ANDNOT 1314.01  ; 关闭#1、#2腔体合模气缸，数据初始化
OUT W221.09  ; #2合模气缸缩回

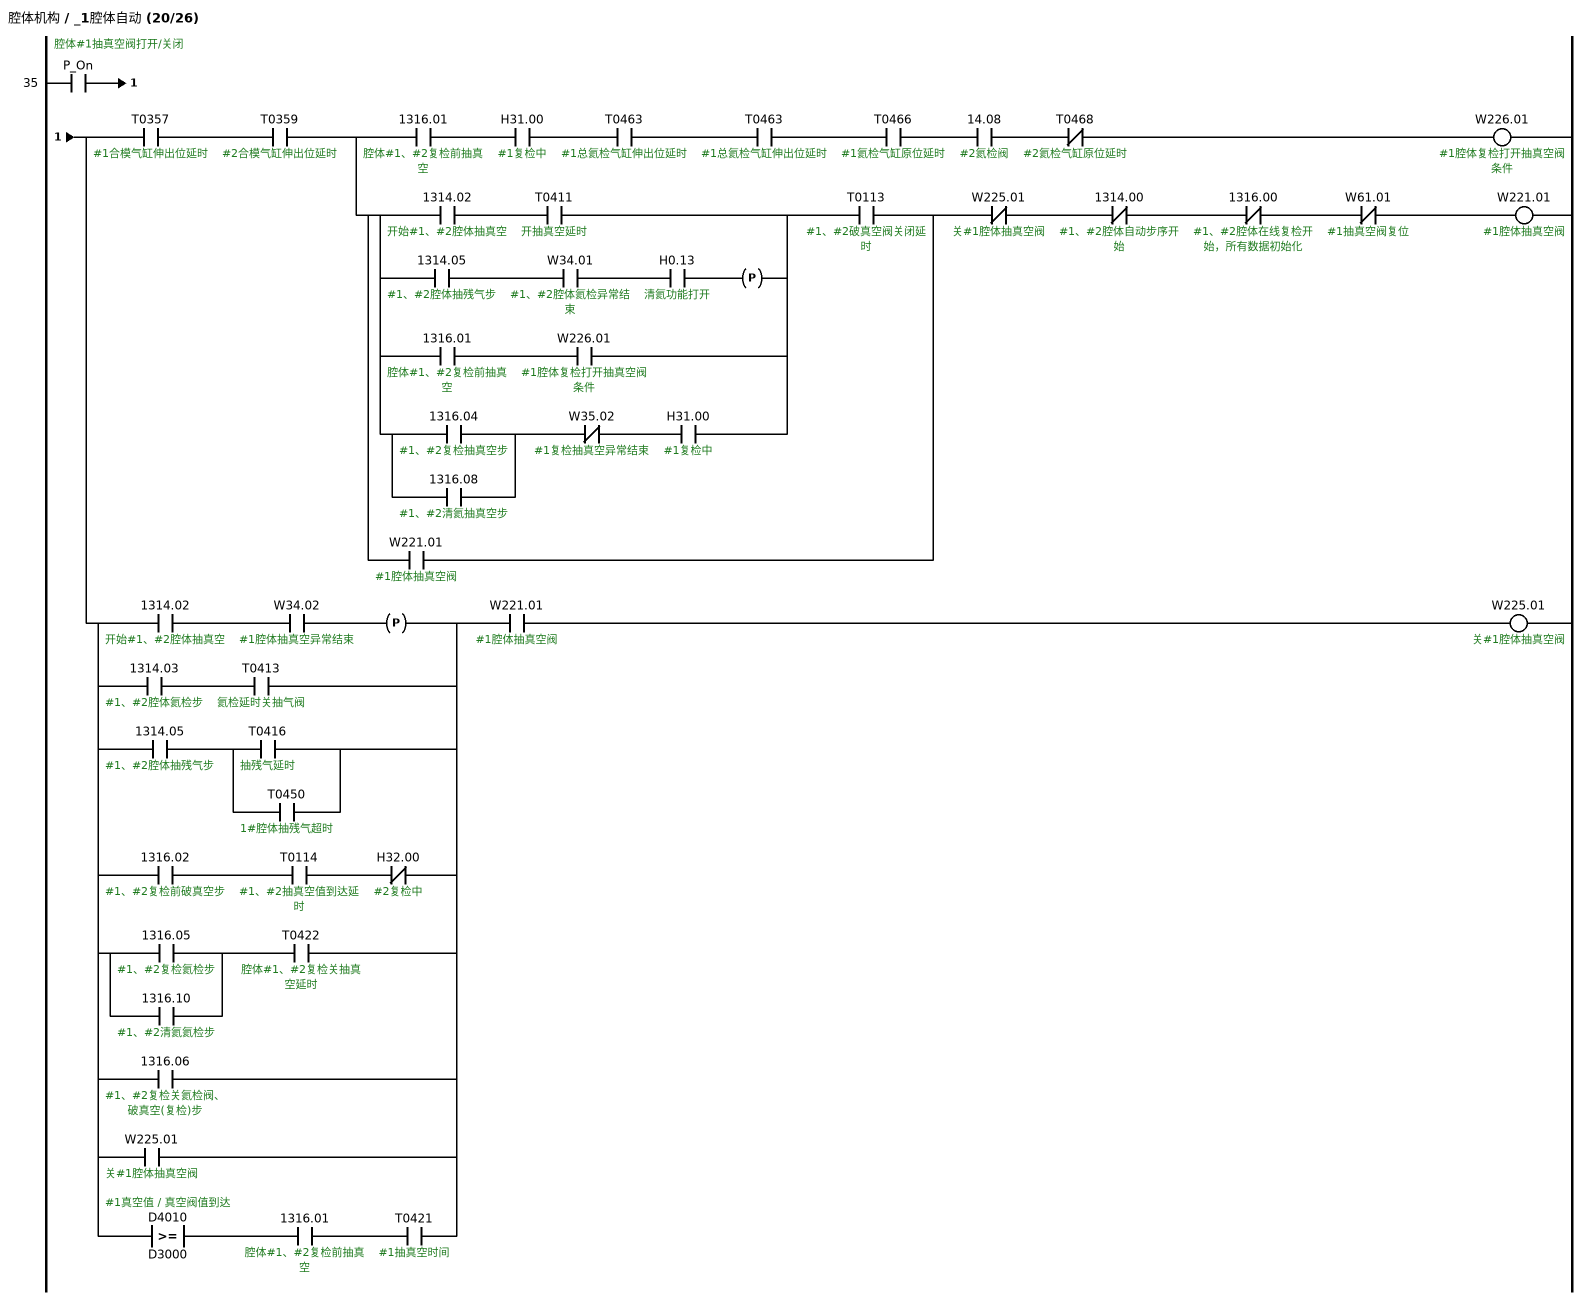
; rung 35: 腔体#1抽真空阀打开/关闭
LD P_On
OUT TR0
AND T0357  ; #1合模气缸伸出位延时
AND T0359  ; #2合模气缸伸出位延时
OUT TR1
AND 1316.01  ; 腔体#1、#2复检前抽真空
AND H31.00  ; #1复检中
AND T0463  ; #1总氦检气缸伸出位延时
AND T0463  ; #1总氦检气缸伸出位延时
AND T0466  ; #1氦检气缸原位延时
AND 14.08  ; #2氦检阀
ANDNOT T0468  ; #2氦检气缸原位延时
OUT W226.01  ; #1腔体复检打开抽真空阀条件
LD TR1
LD 1314.02  ; 开始#1、#2腔体抽真空
AND T0411  ; 开抽真空延时
LD 1314.05  ; #1、#2腔体抽残气步
AND W34.01  ; #1、#2腔体氦检异常结束
AND H0.13  ; 清氦功能打开
UP(521)
ORLD
LD 1316.01  ; 腔体#1、#2复检前抽真空
AND W226.01  ; #1腔体复检打开抽真空阀条件
ORLD
LD 1316.04  ; #1、#2复检抽真空步
OR 1316.08  ; #1、#2清氦抽真空步
ANDNOT W35.02  ; #1复检抽真空异常结束
AND H31.00  ; #1复检中
ORLD
AND T0113  ; #1、#2破真空阀关闭延时
OR W221.01  ; #1腔体抽真空阀
ANDLD
ANDNOT W225.01  ; 关#1腔体抽真空阀
ANDNOT 1314.00  ; #1、#2腔体自动步序开始
ANDNOT 1316.00  ; #1、#2腔体在线复检开始，所有数据初始化
ANDNOT W61.01  ; #1抽真空阀复位
OUT W221.01  ; #1腔体抽真空阀
LD TR0
LD 1314.02  ; 开始#1、#2腔体抽真空
AND W34.02  ; #1腔体抽真空异常结束
UP(521)
LD 1314.03  ; #1、#2腔体氦检步
AND T0413  ; 氦检延时关抽气阀
ORLD
LD 1314.05  ; #1、#2腔体抽残气步
LD T0416  ; 抽残气延时
OR T0450  ; 1#腔体抽残气超时
ANDLD
ORLD
LD 1316.02  ; #1、#2复检前破真空步
AND T0114  ; #1、#2抽真空值到达延时
ANDNOT H32.00  ; #2复检中
ORLD
LD 1316.05  ; #1、#2复检氦检步
OR 1316.10  ; #1、#2清氦氦检步
AND T0422  ; 腔体#1、#2复检关抽真空延时
ORLD
OR 1316.06  ; #1、#2复检关氦检阀、破真空(复检)步
OR W225.01  ; 关#1腔体抽真空阀
LD>=F(334) D4010 D3000  ; #1真空值, 真空阀值到达
AND 1316.01  ; 腔体#1、#2复检前抽真空
AND T0421  ; #1抽真空时间
ORLD
ANDLD
AND W221.01  ; #1腔体抽真空阀
OUT W225.01  ; 关#1腔体抽真空阀

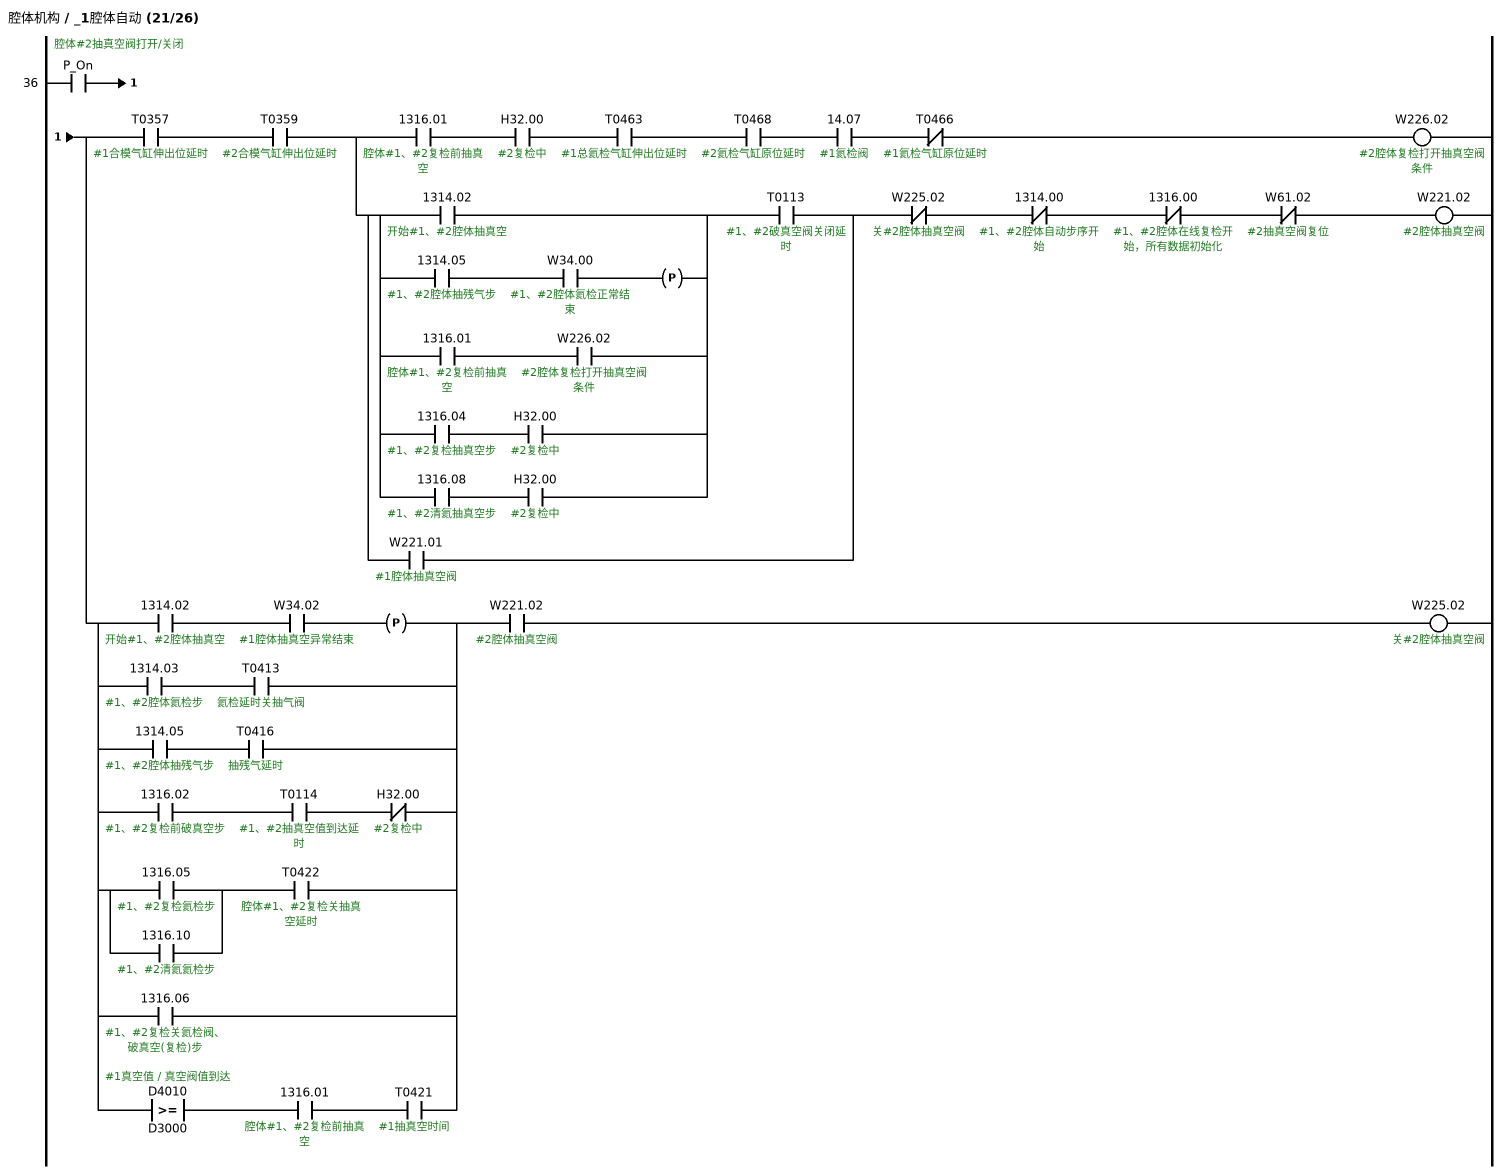
; rung 36: 腔体#2抽真空阀打开/关闭
LD P_On
OUT TR0
AND T0357  ; #1合模气缸伸出位延时
AND T0359  ; #2合模气缸伸出位延时
OUT TR1
AND 1316.01  ; 腔体#1、#2复检前抽真空
AND H32.00  ; #2复检中
AND T0463  ; #1总氦检气缸伸出位延时
AND T0468  ; #2氦检气缸原位延时
AND 14.07  ; #1氦检阀
ANDNOT T0466  ; #1氦检气缸原位延时
OUT W226.02  ; #2腔体复检打开抽真空阀条件
LD TR1
LD 1314.02  ; 开始#1、#2腔体抽真空
LD 1314.05  ; #1、#2腔体抽残气步
AND W34.00  ; #1、#2腔体氦检正常结束
UP(521)
ORLD
LD 1316.01  ; 腔体#1、#2复检前抽真空
AND W226.02  ; #2腔体复检打开抽真空阀条件
ORLD
LD 1316.04  ; #1、#2复检抽真空步
AND H32.00  ; #2复检中
ORLD
LD 1316.08  ; #1、#2清氦抽真空步
AND H32.00  ; #2复检中
ORLD
AND T0113  ; #1、#2破真空阀关闭延时
OR W221.01  ; #1腔体抽真空阀
ANDLD
ANDNOT W225.02  ; 关#2腔体抽真空阀
ANDNOT 1314.00  ; #1、#2腔体自动步序开始
ANDNOT 1316.00  ; #1、#2腔体在线复检开始，所有数据初始化
ANDNOT W61.02  ; #2抽真空阀复位
OUT W221.02  ; #2腔体抽真空阀
LD TR0
LD 1314.02  ; 开始#1、#2腔体抽真空
AND W34.02  ; #1腔体抽真空异常结束
UP(521)
LD 1314.03  ; #1、#2腔体氦检步
AND T0413  ; 氦检延时关抽气阀
ORLD
LD 1314.05  ; #1、#2腔体抽残气步
AND T0416  ; 抽残气延时
ORLD
LD 1316.02  ; #1、#2复检前破真空步
AND T0114  ; #1、#2抽真空值到达延时
ANDNOT H32.00  ; #2复检中
ORLD
LD 1316.05  ; #1、#2复检氦检步
OR 1316.10  ; #1、#2清氦氦检步
AND T0422  ; 腔体#1、#2复检关抽真空延时
ORLD
OR 1316.06  ; #1、#2复检关氦检阀、破真空(复检)步
LD>=F(334) D4010 D3000  ; #1真空值, 真空阀值到达
AND 1316.01  ; 腔体#1、#2复检前抽真空
AND T0421  ; #1抽真空时间
ORLD
ANDLD
AND W221.02  ; #2腔体抽真空阀
OUT W225.02  ; 关#2腔体抽真空阀

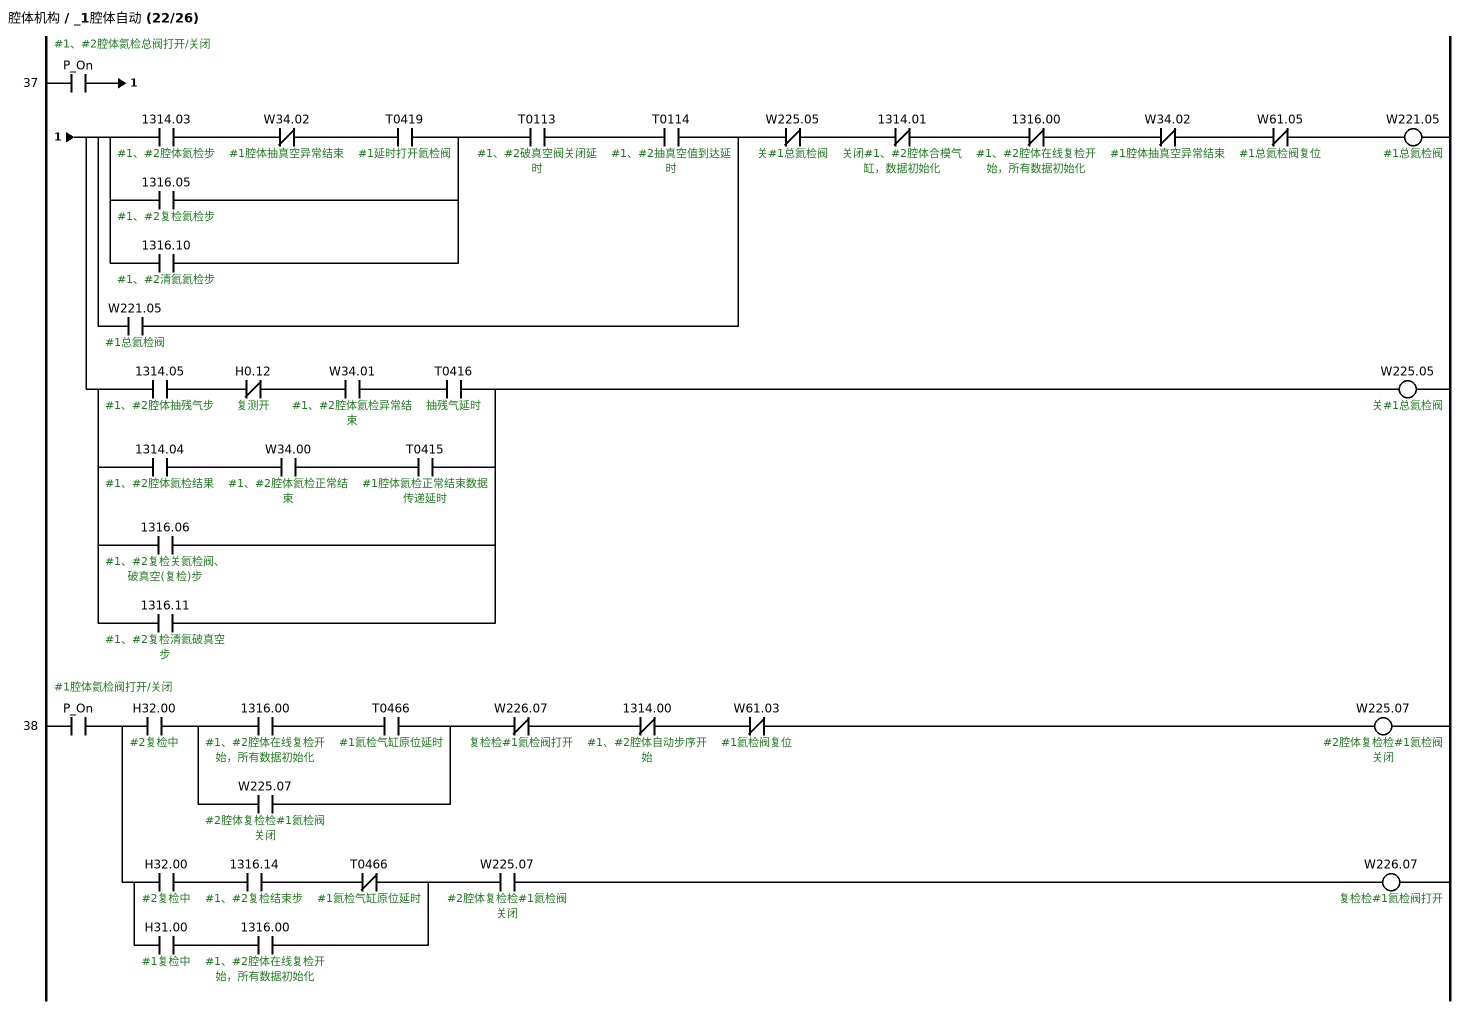
; rung 37: #1、#2腔体氦检总阀打开/关闭
LD P_On
OUT TR0
LD 1314.03  ; #1、#2腔体氦检步
ANDNOT W34.02  ; #1腔体抽真空异常结束
AND T0419  ; #1延时打开氦检阀
OR 1316.05  ; #1、#2复检氦检步
OR 1316.10  ; #1、#2清氦氦检步
AND T0113  ; #1、#2破真空阀关闭延时
AND T0114  ; #1、#2抽真空值到达延时
OR W221.05  ; #1总氦检阀
ANDLD
ANDNOT W225.05  ; 关#1总氦检阀
ANDNOT 1314.01  ; 关闭#1、#2腔体合模气缸，数据初始化
ANDNOT 1316.00  ; #1、#2腔体在线复检开始，所有数据初始化
ANDNOT W34.02  ; #1腔体抽真空异常结束
ANDNOT W61.05  ; #1总氦检阀复位
OUT W221.05  ; #1总氦检阀
LD TR0
LD 1314.05  ; #1、#2腔体抽残气步
ANDNOT H0.12  ; 复测开
AND W34.01  ; #1、#2腔体氦检异常结束
AND T0416  ; 抽残气延时
LD 1314.04  ; #1、#2腔体氦检结果
AND W34.00  ; #1、#2腔体氦检正常结束
AND T0415  ; #1腔体氦检正常结束数据传递延时
ORLD
OR 1316.06  ; #1、#2复检关氦检阀、破真空(复检)步
OR 1316.11  ; #1、#2复检清氦破真空步
ANDLD
OUT W225.05  ; 关#1总氦检阀
; rung 38: #1腔体氦检阀打开/关闭
LD P_On
OUT TR0
AND H32.00  ; #2复检中
LD 1316.00  ; #1、#2腔体在线复检开始，所有数据初始化
AND T0466  ; #1氦检气缸原位延时
OR W225.07  ; #2腔体复检检#1氦检阀关闭
ANDLD
ANDNOT W226.07  ; 复检检#1氦检阀打开
ANDNOT 1314.00  ; #1、#2腔体自动步序开始
ANDNOT W61.03  ; #1氦检阀复位
OUT W225.07  ; #2腔体复检检#1氦检阀关闭
LD TR0
LD H32.00  ; #2复检中
AND 1316.14  ; #1、#2复检结束步
ANDNOT T0466  ; #1氦检气缸原位延时
LD H31.00  ; #1复检中
AND 1316.00  ; #1、#2腔体在线复检开始，所有数据初始化
ORLD
ANDLD
AND W225.07  ; #2腔体复检检#1氦检阀关闭
OUT W226.07  ; 复检检#1氦检阀打开

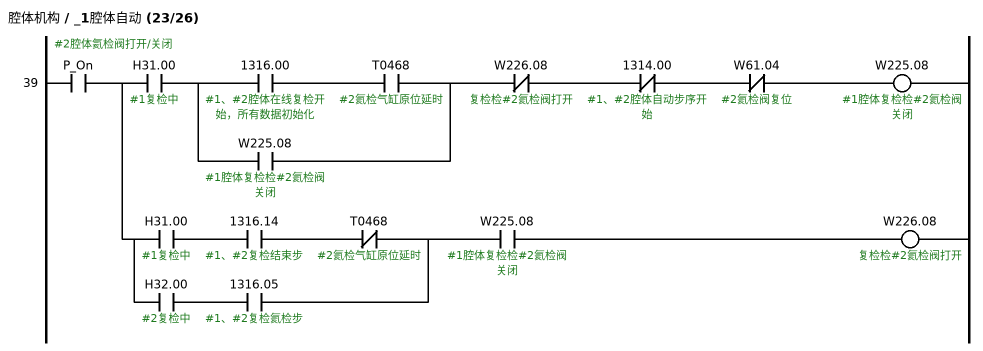
; rung 39: #2腔体氦检阀打开/关闭
LD P_On
OUT TR0
AND H31.00  ; #1复检中
LD 1316.00  ; #1、#2腔体在线复检开始，所有数据初始化
AND T0468  ; #2氦检气缸原位延时
OR W225.08  ; #1腔体复检检#2氦检阀关闭
ANDLD
ANDNOT W226.08  ; 复检检#2氦检阀打开
ANDNOT 1314.00  ; #1、#2腔体自动步序开始
ANDNOT W61.04  ; #2氦检阀复位
OUT W225.08  ; #1腔体复检检#2氦检阀关闭
LD TR0
LD H31.00  ; #1复检中
AND 1316.14  ; #1、#2复检结束步
ANDNOT T0468  ; #2氦检气缸原位延时
LD H32.00  ; #2复检中
AND 1316.05  ; #1、#2复检氦检步
ORLD
ANDLD
AND W225.08  ; #1腔体复检检#2氦检阀关闭
OUT W226.08  ; 复检检#2氦检阀打开

